LIN {X 0,Y 390.064,Z 239.895,A -85,B 0,C 180,E1 -11765.518,E2 -11765.518} C_VEL
LIN {X 0,Y 390.059,Z 239.898,A -85,B 0,C 180,E1 -11768.878,E2 -11768.878} C_VEL
LIN {X 0,Y 390.13,Z 239.89,A -85,B 0,C 180,E1 -11772.167,E2 -11772.167} C_VEL
LIN {X 0,Y 390.147,Z 239.885,A -85,B 0,C 180,E1 -11775.392,E2 -11775.392} C_VEL
LIN {X 0,Y 390.15,Z 239.886,A -85,B 0,C 180,E1 -11778.571,E2 -11778.571} C_VEL
LIN {X 0,Y 390.259,Z 239.876,A -85,B 0,C 180,E1 -11782.086,E2 -11782.086} C_VEL
LIN {X 0,Y 390.199,Z 239.878,A -85,B 0,C 180,E1 -11784.833,E2 -11784.833} C_VEL
LIN {X 0,Y 390.407,Z 239.856,A -85,B 0,C 180,E1 -11787.937,E2 -11787.937} C_VEL
LIN {X 0,Y 390.295,Z 239.866,A -85,B 0,C 180,E1 -11791.032,E2 -11791.032} C_VEL
LIN {X 0,Y 390.263,Z 239.871,A -85,B 0,C 180,E1 -11793.097,E2 -11793.097} C_VEL
LIN {X 0,Y 390.058,Z 240.018,A -85,B 0,C 180,E1 -11795.428,E2 -11795.428} C_VEL
LIN {X 0,Y 389.833,Z 246.867,A -85,B 0,C 180,E1 -11798.815,E2 -11798.815} C_VEL
LIN {X 0,Y 389.754,Z 254.263,A -85,B 0,C 180,E1 -11802.497,E2 -11802.497} C_VEL
LIN {X 0,Y 389.562,Z 261.72,A -85,B 0,C 180,E1 -11806.238,E2 -11806.238} C_VEL
LIN {X 0,Y 389.404,Z 267.139,A -85,B 0,C 180,E1 -11808.957,E2 -11808.957} C_VEL
LIN {X 0,Y 389.348,Z 274.683,A -85,B 0,C 180,E1 -11812.716,E2 -11812.716} C_VEL
LIN {X 0,Y 391.468,Z 286.466,A -85,B 0,C 180,E1 -11813.264,E2 -11813.264} C_VEL
LIN {X 0,Y 391.781,Z 288.367,A -85,B 0,C 180,E1 -11813.369,E2 -11813.369} C_VEL
LIN {X 0,Y 391.491,Z 292.048,A -85,B 0,C 180,E1 -11813.57,E2 -11813.57} C_VEL
LIN {X 0,Y 390.029,Z 295.619,A -85,B 0,C 180,E1 -11813.741,E2 -11813.741} C_VEL
LIN {X 0,Y 385.706,Z 303.652,A -85,B 0,C 180,E1 -11814.196,E2 -11814.196} C_VEL
LIN {X 0,Y 384.887,Z 307.067,A -85,B 0,C 180,E1 -11814.478,E2 -11814.478} C_VEL
LIN {X 0,Y 384.4,Z 315.281,A -85,B 0,C 180,E1 -11815.3,E2 -11815.3} C_VEL
LIN {X 0,Y 383.946,Z 322.929,A -85,B 0,C 180,E1 -11816.242,E2 -11816.242} C_VEL
LIN {X 0,Y 383.463,Z 329.813,A -85,B 0,C 180,E1 -11817.271,E2 -11817.271} C_VEL
LIN {X 0,Y 382.862,Z 337.958,A -85,B 0,C 180,E1 -11818.807,E2 -11818.807} C_VEL
LIN {X 0,Y 382.577,Z 341.952,A -85,B 0,C 180,E1 -11819.735,E2 -11819.735} C_VEL
LIN {X 0,Y 382.282,Z 346.3,A -85,B 0,C 180,E1 -11820.982,E2 -11820.982} C_VEL
LIN {X 0,Y 382.017,Z 349.759,A -85,B 0,C 180,E1 -11822.243,E2 -11822.243} C_VEL
LIN {X 0,Y 381.771,Z 353.226,A -85,B 0,C 180,E1 -11824.064,E2 -11824.064} C_VEL
LIN {X 0,Y 381.621,Z 355.211,A -85,B 0,C 180,E1 -11825.873,E2 -11825.873} C_VEL
LIN {X 0,Y 381.614,Z 355.585,A -85,B 0,C 180,E1 -11827.635,E2 -11827.635} C_VEL
LIN {X 0,Y 381.705,Z 354.659,A -85,B 0,C 180,E1 -11829.348,E2 -11829.348} C_VEL
LIN {X 0,Y 381.96,Z 352.506,A -85,B 0,C 180,E1 -11831.027,E2 -11831.027} C_VEL
LIN {X 0,Y 382.337,Z 348.46,A -85,B 0,C 180,E1 -11832.853,E2 -11832.853} C_VEL
LIN {X 0,Y 382.689,Z 344.128,A -85,B 0,C 180,E1 -11834.256,E2 -11834.256} C_VEL
LIN {X 0,Y 383.166,Z 338.499,A -85,B 0,C 180,E1 -11835.671,E2 -11835.671} C_VEL
LIN {X 0,Y 383.79,Z 331.204,A -85,B 0,C 180,E1 -11837.095,E2 -11837.095} C_VEL
LIN {X 0,Y 384.405,Z 323.923,A -85,B 0,C 180,E1 -11838.211,E2 -11838.211} C_VEL
LIN {X 0,Y 384.9,Z 317.284,A -85,B 0,C 180,E1 -11839.056,E2 -11839.056} C_VEL
LIN {X 0,Y 385.39,Z 310.045,A -85,B 0,C 180,E1 -11839.823,E2 -11839.823} C_VEL
LIN {X 0,Y 385.892,Z 301.292,A -85,B 0,C 180,E1 -11840.573,E2 -11840.573} C_VEL
LIN {X 0,Y 386.17,Z 294.889,A -85,B 0,C 180,E1 -11841.022,E2 -11841.022} C_VEL
LIN {X 0,Y 384.636,Z 285.462,A -85,B 0,C 180,E1 -11841.622,E2 -11841.622} C_VEL
LIN {X 0,Y 382.519,Z 275.828,A -85,B 0,C 180,E1 -11842.116,E2 -11842.116} C_VEL
LIN {X 0,Y 382.655,Z 268.589,A -85,B 0,C 180,E1 -11845.74,E2 -11845.74} C_VEL
LIN {X 0,Y 382.785,Z 261.93,A -85,B 0,C 180,E1 -11849.063,E2 -11849.063} C_VEL
LIN {X 0,Y 382.923,Z 256.534,A -85,B 0,C 180,E1 -11851.76,E2 -11851.76} C_VEL
LIN {X 0,Y 383.075,Z 248.588,A -85,B 0,C 180,E1 -11855.619,E2 -11855.619} C_VEL
LIN {X 0,Y 383.186,Z 242.55,A -85,B 0,C 180,E1 -11858.48,E2 -11858.48} C_VEL
LIN {X 0,Y 383.007,Z 240.78,A -85,B 0,C 180,E1 -11859.363,E2 -11859.363} C_VEL
LIN {X 0,Y 383.107,Z 240.766,A -85,B 0,C 180,E1 -11862.931,E2 -11862.931} C_VEL
LIN {X 0,Y 383.128,Z 240.763,A -85,B 0,C 180,E1 -11866.464,E2 -11866.464} C_VEL
LIN {X 0,Y 383.154,Z 240.762,A -85,B 0,C 180,E1 -11870.498,E2 -11870.498} C_VEL
LIN {X 0,Y 383.246,Z 240.748,A -85,B 0,C 180,E1 -11873.683,E2 -11873.683} C_VEL
LIN {X 0,Y 383.388,Z 240.73,A -85,B 0,C 180,E1 -11877.899,E2 -11877.899} C_VEL
LIN {X 0,Y 383.52,Z 240.713,A -85,B 0,C 180,E1 -11880,E2 -11880} C_VEL
LIN {X 0,Y 383.248,Z 240.747,A -85,B 0,C 180,E1 -11883.154,E2 -11883.154} C_VEL
LIN {X 0,Y 383.258,Z 240.745,A -85,B 0,C 180,E1 -11886.317,E2 -11886.317} C_VEL
LIN {X 0,Y 383.153,Z 240.76,A -85,B 0,C 180,E1 -11889.502,E2 -11889.502} C_VEL
LIN {X 0,Y 383.127,Z 240.76,A -85,B 0,C 180,E1 -11893.536,E2 -11893.536} C_VEL
LIN {X 0,Y 383.097,Z 240.766,A -85,B 0,C 180,E1 -11897.454,E2 -11897.454} C_VEL
LIN {X 0,Y 383.03,Z 240.773,A -85,B 0,C 180,E1 -11900.647,E2 -11900.647} C_VEL
LIN {X 0,Y 383.023,Z 240.774,A -85,B 0,C 180,E1 -11903.808,E2 -11903.808} C_VEL
LIN {X 0,Y 383.08,Z 240.768,A -85,B 0,C 180,E1 -11906.123,E2 -11906.123} C_VEL
LIN {X 0,Y 383.042,Z 240.774,A -85,B 0,C 180,E1 -11908.493,E2 -11908.493} C_VEL
LIN {X 0,Y 383.011,Z 240.774,A -85,B 0,C 180,E1 -11912.15,E2 -11912.15} C_VEL
LIN {X 0,Y 383.019,Z 240.773,A -85,B 0,C 180,E1 -11914.668,E2 -11914.668} C_VEL
LIN {X 0,Y 383.001,Z 240.777,A -85,B 0,C 180,E1 -11917.904,E2 -11917.904} C_VEL
LIN {X 0,Y 382.985,Z 240.78,A -85,B 0,C 180,E1 -11921.347,E2 -11921.347} C_VEL
LIN {X 0,Y 382.997,Z 240.779,A -85,B 0,C 180,E1 -11924.303,E2 -11924.303} C_VEL
LIN {X 0,Y 383.08,Z 240.924,A -85,B 0,C 180,E1 -11926.817,E2 -11926.817} C_VEL
LIN {X 0,Y 384.123,Z 247.016,A -85,B 0,C 180,E1 -11930.214,E2 -11930.214} C_VEL
LIN {X 0,Y 384.988,Z 252.135,A -85,B 0,C 180,E1 -11932.957,E2 -11932.957} C_VEL
LIN {X 0,Y 384.935,Z 256.673,A -85,B 0,C 180,E1 -11935.245,E2 -11935.245} C_VEL
LIN {X 0,Y 384.304,Z 262.28,A -85,B 0,C 180,E1 -11937.971,E2 -11937.971} C_VEL
LIN {X 0,Y 383.595,Z 269.862,A -85,B 0,C 180,E1 -11941.574,E2 -11941.574} C_VEL
LIN {X 0,Y 383.025,Z 277.322,A -85,B 0,C 180,E1 -11945.038,E2 -11945.038} C_VEL
LIN {X 0,Y 382.517,Z 284.78,A -85,B 0,C 180,E1 -11948.441,E2 -11948.441} C_VEL
LIN {X 0,Y 382.133,Z 292.511,A -85,B 0,C 180,E1 -11951.92,E2 -11951.92} C_VEL
LIN {X 0,Y 383.821,Z 306.099,A -85,B 0,C 180,E1 -11952.506,E2 -11952.506} C_VEL
LIN {X 0,Y 385.335,Z 319.619,A -85,B 0,C 180,E1 -11953.306,E2 -11953.306} C_VEL
LIN {X 0,Y 385.814,Z 325.668,A -85,B 0,C 180,E1 -11953.736,E2 -11953.736} C_VEL
LIN {X 0,Y 384.998,Z 337.028,A -85,B 0,C 180,E1 -11954.651,E2 -11954.651} C_VEL
LIN {X 0,Y 384.223,Z 347.555,A -85,B 0,C 180,E1 -11955.712,E2 -11955.712} C_VEL
LIN {X 0,Y 383.503,Z 358.111,A -85,B 0,C 180,E1 -11957.027,E2 -11957.027} C_VEL
LIN {X 0,Y 382.872,Z 366.826,A -85,B 0,C 180,E1 -11958.351,E2 -11958.351} C_VEL
LIN {X 0,Y 382.323,Z 375.346,A -85,B 0,C 180,E1 -11959.943,E2 -11959.943} C_VEL
LIN {X 0,Y 382.009,Z 382.192,A -85,B 0,C 180,E1 -11961.537,E2 -11961.537} C_VEL
LIN {X 0,Y 381.83,Z 387.648,A -85,B 0,C 180,E1 -11963.129,E2 -11963.129} C_VEL
LIN {X 0,Y 381.746,Z 391.876,A -85,B 0,C 180,E1 -11964.719,E2 -11964.719} C_VEL
LIN {X 0,Y 381.68,Z 394.089,A -85,B 0,C 180,E1 -11965.776,E2 -11965.776} C_VEL
LIN {X 0,Y 381.711,Z 395.798,A -85,B 0,C 180,E1 -11966.834,E2 -11966.834} C_VEL
LIN {X 0,Y 381.784,Z 397.076,A -85,B 0,C 180,E1 -11967.89,E2 -11967.89} C_VEL
LIN {X 0,Y 381.741,Z 397.928,A -85,B 0,C 180,E1 -11968.945,E2 -11968.945} C_VEL
LIN {X 0,Y 381.728,Z 398.341,A -85,B 0,C 180,E1 -11970,E2 -11970} C_VEL
LIN {X 0,Y 381.722,Z 398.306,A -85,B 0,C 180,E1 -11971.055,E2 -11971.055} C_VEL
LIN {X 0,Y 381.745,Z 397.863,A -85,B 0,C 180,E1 -11972.11,E2 -11972.11} C_VEL
LIN {X 0,Y 381.625,Z 397.006,A -85,B 0,C 180,E1 -11973.167,E2 -11973.167} C_VEL
LIN {X 0,Y 381.653,Z 395.705,A -85,B 0,C 180,E1 -11974.224,E2 -11974.224} C_VEL
LIN {X 0,Y 381.69,Z 392.269,A -85,B 0,C 180,E1 -11976.122,E2 -11976.122} C_VEL
LIN {X 0,Y 381.912,Z 387.634,A -85,B 0,C 180,E1 -11977.933,E2 -11977.933} C_VEL
LIN {X 0,Y 382.365,Z 381.352,A -85,B 0,C 180,E1 -11979.789,E2 -11979.789} C_VEL
LIN {X 0,Y 383.047,Z 373.281,A -85,B 0,C 180,E1 -11981.644,E2 -11981.644} C_VEL
LIN {X 0,Y 384.014,Z 364.697,A -85,B 0,C 180,E1 -11983.225,E2 -11983.225} C_VEL
LIN {X 0,Y 384.9,Z 355.689,A -85,B 0,C 180,E1 -11984.592,E2 -11984.592} C_VEL
LIN {X 0,Y 386.269,Z 344.532,A -85,B 0,C 180,E1 -11985.974,E2 -11985.974} C_VEL
LIN {X 0,Y 387.633,Z 332.921,A -85,B 0,C 180,E1 -11987.135,E2 -11987.135} C_VEL
LIN {X 0,Y 388.132,Z 325.333,A -85,B 0,C 180,E1 -11987.792,E2 -11987.792} C_VEL
LIN {X 0,Y 387.528,Z 312.932,A -85,B 0,C 180,E1 -11988.781,E2 -11988.781} C_VEL
LIN {X 0,Y 385.488,Z 300.133,A -85,B 0,C 180,E1 -11989.711,E2 -11989.711} C_VEL
LIN {X 0,Y 382.494,Z 287.785,A -85,B 0,C 180,E1 -11990.559,E2 -11990.559} C_VEL
LIN {X 0,Y 382.921,Z 280.937,A -85,B 0,C 180,E1 -11993.815,E2 -11993.815} C_VEL
LIN {X 0,Y 383.578,Z 274.157,A -85,B 0,C 180,E1 -11997.262,E2 -11997.262} C_VEL
LIN {X 0,Y 384.413,Z 267.801,A -85,B 0,C 180,E1 -12000.791,E2 -12000.791} C_VEL
LIN {X 0,Y 385.452,Z 262.026,A -85,B 0,C 180,E1 -12004.418,E2 -12004.418} C_VEL
LIN {X 0,Y 385.784,Z 258.61,A -85,B 0,C 180,E1 -12006.955,E2 -12006.955} C_VEL
LIN {X 0,Y 385.601,Z 255.652,A -85,B 0,C 180,E1 -12009.637,E2 -12009.637} C_VEL
LIN {X 0,Y 385.196,Z 253.221,A -85,B 0,C 180,E1 -12012.461,E2 -12012.461} C_VEL
LIN {X 0,Y 384.881,Z 251.375,A -85,B 0,C 180,E1 -12015.41,E2 -12015.41} C_VEL
LIN {X 0,Y 384.65,Z 250.149,A -85,B 0,C 180,E1 -12018.515,E2 -12018.515} C_VEL
LIN {X 0,Y 384.459,Z 249.598,A -85,B 0,C 180,E1 -12021.819,E2 -12021.819} C_VEL
LIN {X 0,Y 384.362,Z 249.644,A -85,B 0,C 180,E1 -12024.189,E2 -12024.189} C_VEL
LIN {X 0,Y 384.031,Z 250.218,A -85,B 0,C 180,E1 -12027.334,E2 -12027.334} C_VEL
LIN {X 0,Y 383.652,Z 251.212,A -85,B 0,C 180,E1 -12030.356,E2 -12030.356} C_VEL
LIN {X 0,Y 383.284,Z 252.849,A -85,B 0,C 180,E1 -12033.96,E2 -12033.96} C_VEL
LIN {X 0,Y 382.967,Z 254.746,A -85,B 0,C 180,E1 -12037.333,E2 -12037.333} C_VEL
LIN {X 0,Y 382.794,Z 256.871,A -85,B 0,C 180,E1 -12040.633,E2 -12040.633} C_VEL
LIN {X 0,Y 383.82,Z 259.798,A -85,B 0,C 180,E1 -12040.87,E2 -12040.87} C_VEL
LIN {X 0,Y 387.985,Z 270.603,A -85,B 0,C 180,E1 -12041.849,E2 -12041.849} C_VEL
LIN {X 0,Y 390.513,Z 280.022,A -85,B 0,C 180,E1 -12042.712,E2 -12042.712} C_VEL
LIN {X 0,Y 390.497,Z 283.446,A -85,B 0,C 180,E1 -12042.977,E2 -12042.977} C_VEL
LIN {X 0,Y 389.314,Z 295.932,A -85,B 0,C 180,E1 -12044.029,E2 -12044.029} C_VEL
LIN {X 0,Y 388.056,Z 306.9,A -85,B 0,C 180,E1 -12045.178,E2 -12045.178} C_VEL
LIN {X 0,Y 386.93,Z 315.954,A -85,B 0,C 180,E1 -12046.342,E2 -12046.342} C_VEL
LIN {X 0,Y 385.714,Z 325.894,A -85,B 0,C 180,E1 -12047.905,E2 -12047.905} C_VEL
LIN {X 0,Y 384.598,Z 333.903,A -85,B 0,C 180,E1 -12049.471,E2 -12049.471} C_VEL
LIN {X 0,Y 383.857,Z 340.374,A -85,B 0,C 180,E1 -12051.047,E2 -12051.047} C_VEL
LIN {X 0,Y 383.015,Z 345.589,A -85,B 0,C 180,E1 -12052.62,E2 -12052.62} C_VEL
LIN {X 0,Y 382.778,Z 349.616,A -85,B 0,C 180,E1 -12054.204,E2 -12054.204} C_VEL
LIN {X 0,Y 382.457,Z 352.63,A -85,B 0,C 180,E1 -12055.785,E2 -12055.785} C_VEL
LIN {X 0,Y 382.34,Z 354.101,A -85,B 0,C 180,E1 -12056.839,E2 -12056.839} C_VEL
LIN {X 0,Y 382.016,Z 355.174,A -85,B 0,C 180,E1 -12057.891,E2 -12057.891} C_VEL
LIN {X 0,Y 381.771,Z 356.022,A -85,B 0,C 180,E1 -12060,E2 -12060} C_VEL
LIN {X 0,Y 381.76,Z 355.851,A -85,B 0,C 180,E1 -12061.055,E2 -12061.055} C_VEL
LIN {X 0,Y 381.827,Z 355.248,A -85,B 0,C 180,E1 -12062.11,E2 -12062.11} C_VEL
LIN {X 0,Y 381.849,Z 354.219,A -85,B 0,C 180,E1 -12063.165,E2 -12063.165} C_VEL
LIN {X 0,Y 381.825,Z 352.79,A -85,B 0,C 180,E1 -12064.222,E2 -12064.222} C_VEL
LIN {X 0,Y 382.002,Z 349.805,A -85,B 0,C 180,E1 -12065.808,E2 -12065.808} C_VEL
LIN {X 0,Y 382.153,Z 345.762,A -85,B 0,C 180,E1 -12067.397,E2 -12067.397} C_VEL
LIN {X 0,Y 382.544,Z 339.557,A -85,B 0,C 180,E1 -12069.251,E2 -12069.251} C_VEL
LIN {X 0,Y 382.976,Z 332.754,A -85,B 0,C 180,E1 -12070.842,E2 -12070.842} C_VEL
LIN {X 0,Y 383.602,Z 324.348,A -85,B 0,C 180,E1 -12072.432,E2 -12072.432} C_VEL
LIN {X 0,Y 384.278,Z 314.547,A -85,B 0,C 180,E1 -12073.924,E2 -12073.924} C_VEL
LIN {X 0,Y 384.893,Z 304.111,A -85,B 0,C 180,E1 -12075.218,E2 -12075.218} C_VEL
LIN {X 0,Y 385.693,Z 293.658,A -85,B 0,C 180,E1 -12076.27,E2 -12076.27} C_VEL
LIN {X 0,Y 386.513,Z 280.873,A -85,B 0,C 180,E1 -12077.289,E2 -12077.289} C_VEL
LIN {X 0,Y 386.737,Z 275.385,A -85,B 0,C 180,E1 -12077.655,E2 -12077.655} C_VEL
LIN {X 0,Y 384.045,Z 262.022,A -85,B 0,C 180,E1 -12078.479,E2 -12078.479} C_VEL
LIN {X 0,Y 381.923,Z 251.524,A -85,B 0,C 180,E1 -12078.994,E2 -12078.994} C_VEL
LIN {X 0,Y 381.915,Z 247.631,A -85,B 0,C 180,E1 -12082.734,E2 -12082.734} C_VEL
LIN {X 0,Y 382.077,Z 244.102,A -85,B 0,C 180,E1 -12086.197,E2 -12086.197} C_VEL
LIN {X 0,Y 382.103,Z 241.747,A -85,B 0,C 180,E1 -12088.569,E2 -12088.569} C_VEL
LIN {X 0,Y 382.166,Z 240.883,A -85,B 0,C 180,E1 -12089.771,E2 -12089.771} C_VEL
LIN {X 0,Y 382.621,Z 240.827,A -85,B 0,C 180,E1 -12093.439,E2 -12093.439} C_VEL
LIN {X 0,Y 382.905,Z 240.787,A -85,B 0,C 180,E1 -12096.138,E2 -12096.138} C_VEL
LIN {X 0,Y 382.996,Z 240.777,A -85,B 0,C 180,E1 -12098.602,E2 -12098.602} C_VEL
LIN {X 0,Y 382.985,Z 240.781,A -85,B 0,C 180,E1 -12101.348,E2 -12101.348} C_VEL
LIN {X 0,Y 382.999,Z 240.775,A -85,B 0,C 180,E1 -12104.303,E2 -12104.303} C_VEL
LIN {X 0,Y 383.014,Z 240.776,A -85,B 0,C 180,E1 -12107.24,E2 -12107.24} C_VEL
LIN {X 0,Y 382.988,Z 240.778,A -85,B 0,C 180,E1 -12110.419,E2 -12110.419} C_VEL
LIN {X 0,Y 383.016,Z 240.772,A -85,B 0,C 180,E1 -12114.043,E2 -12114.043} C_VEL
LIN {X 0,Y 382.989,Z 240.776,A -85,B 0,C 180,E1 -12117.578,E2 -12117.578} C_VEL
LIN {X 0,Y 382.988,Z 240.779,A -85,B 0,C 180,E1 -12120.299,E2 -12120.299} C_VEL
LIN {X 0,Y 383.046,Z 240.771,A -85,B 0,C 180,E1 -12124.032,E2 -12124.032} C_VEL
LIN {X 0,Y 382.995,Z 240.776,A -85,B 0,C 180,E1 -12127.334,E2 -12127.334} C_VEL
LIN {X 0,Y 383.062,Z 240.77,A -85,B 0,C 180,E1 -12130.716,E2 -12130.716} C_VEL
LIN {X 0,Y 383.084,Z 240.768,A -85,B 0,C 180,E1 -12134.027,E2 -12134.027} C_VEL
LIN {X 0,Y 383.14,Z 240.758,A -85,B 0,C 180,E1 -12137.284,E2 -12137.284} C_VEL
LIN {X 0,Y 383.146,Z 240.758,A -85,B 0,C 180,E1 -12140.498,E2 -12140.498} C_VEL
LIN {X 0,Y 383.234,Z 240.748,A -85,B 0,C 180,E1 -12143.683,E2 -12143.683} C_VEL
LIN {X 0,Y 383.371,Z 240.733,A -85,B 0,C 180,E1 -12147.899,E2 -12147.899} C_VEL
LIN {X 0,Y 383.266,Z 240.741,A -85,B 0,C 180,E1 -12151.051,E2 -12151.051} C_VEL
LIN {X 0,Y 383.381,Z 240.729,A -85,B 0,C 180,E1 -12152.101,E2 -12152.101} C_VEL
LIN {X 0,Y 383.049,Z 240.859,A -85,B 0,C 180,E1 -12155.329,E2 -12155.329} C_VEL
LIN {X 0,Y 382.786,Z 248.186,A -85,B 0,C 180,E1 -12158.978,E2 -12158.978} C_VEL
LIN {X 0,Y 382.71,Z 255.662,A -85,B 0,C 180,E1 -12162.73,E2 -12162.73} C_VEL
LIN {X 0,Y 382.488,Z 263.248,A -85,B 0,C 180,E1 -12166.547,E2 -12166.547} C_VEL
LIN {X 0,Y 382.329,Z 269.769,A -85,B 0,C 180,E1 -12169.838,E2 -12169.838} C_VEL
LIN {X 0,Y 382.277,Z 274.974,A -85,B 0,C 180,E1 -12172.461,E2 -12172.461} C_VEL
LIN {X 0,Y 384.76,Z 288.83,A -85,B 0,C 180,E1 -12173.151,E2 -12173.151} C_VEL
LIN {X 0,Y 385.45,Z 294.606,A -85,B 0,C 180,E1 -12173.524,E2 -12173.524} C_VEL
LIN {X 0,Y 384.959,Z 305.487,A -85,B 0,C 180,E1 -12174.332,E2 -12174.332} C_VEL
LIN {X 0,Y 384.887,Z 307.067,A -85,B 0,C 180,E1 -12174.478,E2 -12174.478} C_VEL
LIN {X 0,Y 384.053,Z 312.121,A -85,B 0,C 180,E1 -12174.932,E2 -12174.932} C_VEL
LIN {X 0,Y 380.771,Z 319.846,A -85,B 0,C 180,E1 -12175.722,E2 -12175.722} C_VEL
LIN {X 0,Y 377.398,Z 327.02,A -85,B 0,C 180,E1 -12176.621,E2 -12176.621} C_VEL
LIN {X 0,Y 376.404,Z 331.043,A -85,B 0,C 180,E1 -12177.26,E2 -12177.26} C_VEL
LIN {X 0,Y 375.794,Z 338.668,A -85,B 0,C 180,E1 -12178.761,E2 -12178.761} C_VEL
LIN {X 0,Y 375.433,Z 343.811,A -85,B 0,C 180,E1 -12180.05,E2 -12180.05} C_VEL
LIN {X 0,Y 375.038,Z 348.777,A -85,B 0,C 180,E1 -12181.648,E2 -12181.648} C_VEL
LIN {X 0,Y 374.854,Z 351.743,A -85,B 0,C 180,E1 -12182.937,E2 -12182.937} C_VEL
LIN {X 0,Y 374.647,Z 354.113,A -85,B 0,C 180,E1 -12184.371,E2 -12184.371} C_VEL
LIN {X 0,Y 374.521,Z 355.737,A -85,B 0,C 180,E1 -12186.205,E2 -12186.205} C_VEL
LIN {X 0,Y 374.526,Z 355.893,A -85,B 0,C 180,E1 -12187.988,E2 -12187.988} C_VEL
LIN {X 0,Y 374.662,Z 354.788,A -85,B 0,C 180,E1 -12189.727,E2 -12189.727} C_VEL
LIN {X 0,Y 374.975,Z 352.348,A -85,B 0,C 180,E1 -12191.435,E2 -12191.435} C_VEL
LIN {X 0,Y 375.173,Z 350.351,A -85,B 0,C 180,E1 -12192.406,E2 -12192.406} C_VEL
LIN {X 0,Y 375.501,Z 346.538,A -85,B 0,C 180,E1 -12193.829,E2 -12193.829} C_VEL
LIN {X 0,Y 375.968,Z 341.421,A -85,B 0,C 180,E1 -12195.263,E2 -12195.263} C_VEL
LIN {X 0,Y 376.486,Z 336.09,A -85,B 0,C 180,E1 -12196.457,E2 -12196.457} C_VEL
LIN {X 0,Y 377.021,Z 329.555,A -85,B 0,C 180,E1 -12197.651,E2 -12197.651} C_VEL
LIN {X 0,Y 377.644,Z 322.437,A -85,B 0,C 180,E1 -12198.711,E2 -12198.711} C_VEL
LIN {X 0,Y 378.38,Z 313.351,A -85,B 0,C 180,E1 -12199.805,E2 -12199.805} C_VEL
LIN {X 0,Y 378.987,Z 303.249,A -85,B 0,C 180,E1 -12200.734,E2 -12200.734} C_VEL
LIN {X 0,Y 379.367,Z 296.06,A -85,B 0,C 180,E1 -12201.263,E2 -12201.263} C_VEL
LIN {X 0,Y 377.864,Z 286.83,A -85,B 0,C 180,E1 -12201.877,E2 -12201.877} C_VEL
LIN {X 0,Y 375.685,Z 277.189,A -85,B 0,C 180,E1 -12202.387,E2 -12202.387} C_VEL
LIN {X 0,Y 375.496,Z 276.171,A -85,B 0,C 180,E1 -12202.449,E2 -12202.449} C_VEL
LIN {X 0,Y 375.629,Z 269.437,A -85,B 0,C 180,E1 -12205.854,E2 -12205.854} C_VEL
LIN {X 0,Y 375.802,Z 262.494,A -85,B 0,C 180,E1 -12209.346,E2 -12209.346} C_VEL
LIN {X 0,Y 375.977,Z 255.707,A -85,B 0,C 180,E1 -12212.744,E2 -12212.744} C_VEL
LIN {X 0,Y 376.168,Z 248.436,A -85,B 0,C 180,E1 -12216.273,E2 -12216.273} C_VEL
LIN {X 0,Y 376.135,Z 242.637,A -85,B 0,C 180,E1 -12219.106,E2 -12219.106} C_VEL
LIN {X 0,Y 375.989,Z 241.654,A -85,B 0,C 180,E1 -12219.626,E2 -12219.626} C_VEL
LIN {X 0,Y 376.053,Z 241.645,A -85,B 0,C 180,E1 -12222.601,E2 -12222.601} C_VEL
LIN {X 0,Y 376.092,Z 241.639,A -85,B 0,C 180,E1 -12226.342,E2 -12226.342} C_VEL
LIN {X 0,Y 376.121,Z 241.637,A -85,B 0,C 180,E1 -12230.318,E2 -12230.318} C_VEL
LIN {X 0,Y 376.204,Z 241.625,A -85,B 0,C 180,E1 -12233.564,E2 -12233.564} C_VEL
LIN {X 0,Y 376.354,Z 241.606,A -85,B 0,C 180,E1 -12237.859,E2 -12237.859} C_VEL
LIN {X 0,Y 376.49,Z 241.589,A -85,B 0,C 180,E1 -12240,E2 -12240} C_VEL
LIN {X 0,Y 376.186,Z 241.627,A -85,B 0,C 180,E1 -12243.213,E2 -12243.213} C_VEL
LIN {X 0,Y 376.216,Z 241.623,A -85,B 0,C 180,E1 -12246.435,E2 -12246.435} C_VEL
LIN {X 0,Y 376.121,Z 241.637,A -85,B 0,C 180,E1 -12249.681,E2 -12249.681} C_VEL
LIN {X 0,Y 376.091,Z 241.636,A -85,B 0,C 180,E1 -12253.658,E2 -12253.658} C_VEL
LIN {X 0,Y 376.045,Z 241.645,A -85,B 0,C 180,E1 -12257.607,E2 -12257.607} C_VEL
LIN {X 0,Y 375.98,Z 241.651,A -85,B 0,C 180,E1 -12260.832,E2 -12260.832} C_VEL
LIN {X 0,Y 375.988,Z 241.649,A -85,B 0,C 180,E1 -12264.282,E2 -12264.282} C_VEL
LIN {X 0,Y 376.021,Z 241.644,A -85,B 0,C 180,E1 -12266.652,E2 -12266.652} C_VEL
LIN {X 0,Y 375.972,Z 241.651,A -85,B 0,C 180,E1 -12269.079,E2 -12269.079} C_VEL
LIN {X 0,Y 375.95,Z 241.655,A -85,B 0,C 180,E1 -12272.828,E2 -12272.828} C_VEL
LIN {X 0,Y 375.959,Z 241.653,A -85,B 0,C 180,E1 -12275.415,E2 -12275.415} C_VEL
LIN {X 0,Y 375.976,Z 241.654,A -85,B 0,C 180,E1 -12278.271,E2 -12278.271} C_VEL
LIN {X 0,Y 375.936,Z 241.657,A -85,B 0,C 180,E1 -12281.601,E2 -12281.601} C_VEL
LIN {X 0,Y 375.928,Z 241.661,A -85,B 0,C 180,E1 -12285.269,E2 -12285.269} C_VEL
LIN {X 0,Y 376.035,Z 241.86,A -85,B 0,C 180,E1 -12286.63,E2 -12286.63} C_VEL
LIN {X 0,Y 377.007,Z 247.483,A -85,B 0,C 180,E1 -12289.845,E2 -12289.845} C_VEL
LIN {X 0,Y 377.986,Z 253.43,A -85,B 0,C 180,E1 -12293.084,E2 -12293.084} C_VEL
LIN {X 0,Y 377.933,Z 256.968,A -85,B 0,C 180,E1 -12294.907,E2 -12294.907} C_VEL
LIN {X 0,Y 377.263,Z 263.047,A -85,B 0,C 180,E1 -12297.932,E2 -12297.932} C_VEL
LIN {X 0,Y 376.602,Z 269.964,A -85,B 0,C 180,E1 -12301.294,E2 -12301.294} C_VEL
LIN {X 0,Y 375.931,Z 278.047,A -85,B 0,C 180,E1 -12305.125,E2 -12305.125} C_VEL
LIN {X 0,Y 375.422,Z 285.482,A -85,B 0,C 180,E1 -12308.59,E2 -12308.59} C_VEL
LIN {X 0,Y 375.062,Z 292.213,A -85,B 0,C 180,E1 -12311.686,E2 -12311.686} C_VEL
LIN {X 0,Y 376.724,Z 305.829,A -85,B 0,C 180,E1 -12312.288,E2 -12312.288} C_VEL
LIN {X 0,Y 378.24,Z 319.594,A -85,B 0,C 180,E1 -12313.123,E2 -12313.123} C_VEL
LIN {X 0,Y 378.798,Z 325.628,A -85,B 0,C 180,E1 -12313.564,E2 -12313.564} C_VEL
LIN {X 0,Y 377.968,Z 336.889,A -85,B 0,C 180,E1 -12314.497,E2 -12314.497} C_VEL
LIN {X 0,Y 377.184,Z 347.419,A -85,B 0,C 180,E1 -12315.587,E2 -12315.587} C_VEL
LIN {X 0,Y 376.536,Z 356.896,A -85,B 0,C 180,E1 -12316.783,E2 -12316.783} C_VEL
LIN {X 0,Y 375.879,Z 365.733,A -85,B 0,C 180,E1 -12318.131,E2 -12318.131} C_VEL
LIN {X 0,Y 375.259,Z 374.406,A -85,B 0,C 180,E1 -12319.751,E2 -12319.751} C_VEL
LIN {X 0,Y 374.946,Z 381.347,A -85,B 0,C 180,E1 -12321.376,E2 -12321.376} C_VEL
LIN {X 0,Y 374.748,Z 386.89,A -85,B 0,C 180,E1 -12322.998,E2 -12322.998} C_VEL
LIN {X 0,Y 374.662,Z 391.201,A -85,B 0,C 180,E1 -12324.618,E2 -12324.618} C_VEL
LIN {X 0,Y 374.614,Z 393.459,A -85,B 0,C 180,E1 -12325.696,E2 -12325.696} C_VEL
LIN {X 0,Y 374.62,Z 395.231,A -85,B 0,C 180,E1 -12326.774,E2 -12326.774} C_VEL
LIN {X 0,Y 374.717,Z 396.542,A -85,B 0,C 180,E1 -12327.85,E2 -12327.85} C_VEL
LIN {X 0,Y 374.672,Z 397.424,A -85,B 0,C 180,E1 -12328.925,E2 -12328.925} C_VEL
LIN {X 0,Y 374.657,Z 397.892,A -85,B 0,C 180,E1 -12330,E2 -12330} C_VEL
LIN {X 0,Y 374.654,Z 397.897,A -85,B 0,C 180,E1 -12331.075,E2 -12331.075} C_VEL
LIN {X 0,Y 374.643,Z 397.482,A -85,B 0,C 180,E1 -12332.15,E2 -12332.15} C_VEL
LIN {X 0,Y 374.534,Z 396.654,A -85,B 0,C 180,E1 -12333.227,E2 -12333.227} C_VEL
LIN {X 0,Y 374.577,Z 395.417,A -85,B 0,C 180,E1 -12334.304,E2 -12334.304} C_VEL
LIN {X 0,Y 374.586,Z 392.413,A -85,B 0,C 180,E1 -12336.071,E2 -12336.071} C_VEL
LIN {X 0,Y 374.768,Z 388.991,A -85,B 0,C 180,E1 -12337.543,E2 -12337.543} C_VEL
LIN {X 0,Y 375.087,Z 384.184,A -85,B 0,C 180,E1 -12339.164,E2 -12339.164} C_VEL
LIN {X 0,Y 375.702,Z 377.011,A -85,B 0,C 180,E1 -12341.055,E2 -12341.055} C_VEL
LIN {X 0,Y 376.668,Z 369.381,A -85,B 0,C 180,E1 -12342.664,E2 -12342.664} C_VEL
LIN {X 0,Y 377.508,Z 360.595,A -85,B 0,C 180,E1 -12344.198,E2 -12344.198} C_VEL
LIN {X 0,Y 378.894,Z 349.619,A -85,B 0,C 180,E1 -12345.74,E2 -12345.74} C_VEL
LIN {X 0,Y 380.406,Z 338.026,A -85,B 0,C 180,E1 -12347.055,E2 -12347.055} C_VEL
LIN {X 0,Y 381.526,Z 326.689,A -85,B 0,C 180,E1 -12348.111,E2 -12348.111} C_VEL
LIN {X 0,Y 381.031,Z 314.451,A -85,B 0,C 180,E1 -12349.15,E2 -12349.15} C_VEL
LIN {X 0,Y 379.107,Z 301.802,A -85,B 0,C 180,E1 -12350.14,E2 -12350.14} C_VEL
LIN {X 0,Y 376.206,Z 290.22,A -85,B 0,C 180,E1 -12351.001,E2 -12351.001} C_VEL
LIN {X 0,Y 375.53,Z 287.172,A -85,B 0,C 180,E1 -12351.217,E2 -12351.217} C_VEL
LIN {X 0,Y 376.066,Z 279.805,A -85,B 0,C 180,E1 -12354.866,E2 -12354.866} C_VEL
LIN {X 0,Y 376.662,Z 274.263,A -85,B 0,C 180,E1 -12357.805,E2 -12357.805} C_VEL
LIN {X 0,Y 377.582,Z 268.038,A -85,B 0,C 180,E1 -12361.411,E2 -12361.411} C_VEL
LIN {X 0,Y 378.27,Z 264.222,A -85,B 0,C 180,E1 -12363.875,E2 -12363.875} C_VEL
LIN {X 0,Y 378.798,Z 260.73,A -85,B 0,C 180,E1 -12366.421,E2 -12366.421} C_VEL
LIN {X 0,Y 378.711,Z 257.685,A -85,B 0,C 180,E1 -12369.122,E2 -12369.122} C_VEL
LIN {X 0,Y 378.329,Z 255.129,A -85,B 0,C 180,E1 -12372.007,E2 -12372.007} C_VEL
LIN {X 0,Y 377.995,Z 253.131,A -85,B 0,C 180,E1 -12375.047,E2 -12375.047} C_VEL
LIN {X 0,Y 377.747,Z 251.827,A -85,B 0,C 180,E1 -12378.091,E2 -12378.091} C_VEL
LIN {X 0,Y 377.533,Z 251.15,A -85,B 0,C 180,E1 -12381.432,E2 -12381.432} C_VEL
LIN {X 0,Y 377.373,Z 251.16,A -85,B 0,C 180,E1 -12384.737,E2 -12384.737} C_VEL
LIN {X 0,Y 377.074,Z 251.603,A -85,B 0,C 180,E1 -12387.282,E2 -12387.282} C_VEL
LIN {X 0,Y 376.758,Z 252.336,A -85,B 0,C 180,E1 -12389.758,E2 -12389.758} C_VEL
LIN {X 0,Y 376.344,Z 253.823,A -85,B 0,C 180,E1 -12393.373,E2 -12393.373} C_VEL
LIN {X 0,Y 375.993,Z 255.674,A -85,B 0,C 180,E1 -12396.888,E2 -12396.888} C_VEL
LIN {X 0,Y 375.837,Z 257.545,A -85,B 0,C 180,E1 -12399.975,E2 -12399.975} C_VEL
LIN {X 0,Y 376.94,Z 260.579,A -85,B 0,C 180,E1 -12400.245,E2 -12400.245} C_VEL
LIN {X 0,Y 381.537,Z 272.393,A -85,B 0,C 180,E1 -12401.392,E2 -12401.392} C_VEL
LIN {X 0,Y 384.142,Z 281.948,A -85,B 0,C 180,E1 -12402.33,E2 -12402.33} C_VEL
LIN {X 0,Y 383.477,Z 291.138,A -85,B 0,C 180,E1 -12403.086,E2 -12403.086} C_VEL
LIN {X 0,Y 382.104,Z 303.135,A -85,B 0,C 180,E1 -12404.259,E2 -12404.259} C_VEL
LIN {X 0,Y 380.688,Z 313.843,A -85,B 0,C 180,E1 -12405.568,E2 -12405.568} C_VEL
LIN {X 0,Y 379.565,Z 322.67,A -85,B 0,C 180,E1 -12406.89,E2 -12406.89} C_VEL
LIN {X 0,Y 378.316,Z 331.347,A -85,B 0,C 180,E1 -12408.48,E2 -12408.48} C_VEL
LIN {X 0,Y 377.287,Z 338.4,A -85,B 0,C 180,E1 -12410.078,E2 -12410.078} C_VEL
LIN {X 0,Y 376.316,Z 344.872,A -85,B 0,C 180,E1 -12411.926,E2 -12411.926} C_VEL
LIN {X 0,Y 375.916,Z 349.222,A -85,B 0,C 180,E1 -12413.559,E2 -12413.559} C_VEL
LIN {X 0,Y 375.628,Z 351.479,A -85,B 0,C 180,E1 -12414.632,E2 -12414.632} C_VEL
LIN {X 0,Y 375.41,Z 353.312,A -85,B 0,C 180,E1 -12415.706,E2 -12415.706} C_VEL
LIN {X 0,Y 375.303,Z 354.73,A -85,B 0,C 180,E1 -12416.78,E2 -12416.78} C_VEL
LIN {X 0,Y 374.949,Z 355.721,A -85,B 0,C 180,E1 -12417.852,E2 -12417.852} C_VEL
LIN {X 0,Y 374.698,Z 356.472,A -85,B 0,C 180,E1 -12420,E2 -12420} C_VEL
LIN {X 0,Y 374.691,Z 356.242,A -85,B 0,C 180,E1 -12421.075,E2 -12421.075} C_VEL
LIN {X 0,Y 374.763,Z 355.563,A -85,B 0,C 180,E1 -12422.15,E2 -12422.15} C_VEL
LIN {X 0,Y 374.754,Z 354.487,A -85,B 0,C 180,E1 -12423.225,E2 -12423.225} C_VEL
LIN {X 0,Y 374.751,Z 353.008,A -85,B 0,C 180,E1 -12424.302,E2 -12424.302} C_VEL
LIN {X 0,Y 374.934,Z 349.927,A -85,B 0,C 180,E1 -12425.918,E2 -12425.918} C_VEL
LIN {X 0,Y 375.088,Z 345.783,A -85,B 0,C 180,E1 -12427.537,E2 -12427.537} C_VEL
LIN {X 0,Y 375.516,Z 339.421,A -85,B 0,C 180,E1 -12429.425,E2 -12429.425} C_VEL
LIN {X 0,Y 375.954,Z 332.499,A -85,B 0,C 180,E1 -12431.047,E2 -12431.047} C_VEL
LIN {X 0,Y 376.632,Z 323.946,A -85,B 0,C 180,E1 -12432.666,E2 -12432.666} C_VEL
LIN {X 0,Y 377.325,Z 313.609,A -85,B 0,C 180,E1 -12434.232,E2 -12434.232} C_VEL
LIN {X 0,Y 378.007,Z 303.309,A -85,B 0,C 180,E1 -12435.502,E2 -12435.502} C_VEL
LIN {X 0,Y 378.926,Z 291,A -85,B 0,C 180,E1 -12436.707,E2 -12436.707} C_VEL
LIN {X 0,Y 379.684,Z 278.602,A -85,B 0,C 180,E1 -12437.667,E2 -12437.667} C_VEL
LIN {X 0,Y 379.312,Z 274.155,A -85,B 0,C 180,E1 -12437.974,E2 -12437.974} C_VEL
LIN {X 0,Y 376.628,Z 260.635,A -85,B 0,C 180,E1 -12438.793,E2 -12438.793} C_VEL
LIN {X 0,Y 374.823,Z 251.878,A -85,B 0,C 180,E1 -12439.226,E2 -12439.226} C_VEL
LIN {X 0,Y 374.821,Z 248.978,A -85,B 0,C 180,E1 -12442.025,E2 -12442.025} C_VEL
LIN {X 0,Y 375.025,Z 245.044,A -85,B 0,C 180,E1 -12445.903,E2 -12445.903} C_VEL
LIN {X 0,Y 375.05,Z 241.847,A -85,B 0,C 180,E1 -12449.158,E2 -12449.158} C_VEL
LIN {X 0,Y 375.495,Z 241.712,A -85,B 0,C 180,E1 -12452.874,E2 -12452.874} C_VEL
LIN {X 0,Y 375.805,Z 241.676,A -85,B 0,C 180,E1 -12455.432,E2 -12455.432} C_VEL
LIN {X 0,Y 375.967,Z 241.651,A -85,B 0,C 180,E1 -12458.268,E2 -12458.268} C_VEL
LIN {X 0,Y 375.936,Z 241.657,A -85,B 0,C 180,E1 -12461.6,E2 -12461.6} C_VEL
LIN {X 0,Y 375.929,Z 241.659,A -85,B 0,C 180,E1 -12465.269,E2 -12465.269} C_VEL
LIN {X 0,Y 375.921,Z 241.658,A -85,B 0,C 180,E1 -12468.402,E2 -12468.402} C_VEL
LIN {X 0,Y 375.955,Z 241.651,A -85,B 0,C 180,E1 -12471.91,E2 -12471.91} C_VEL
LIN {X 0,Y 375.977,Z 241.65,A -85,B 0,C 180,E1 -12475.334,E2 -12475.334} C_VEL
LIN {X 0,Y 375.96,Z 241.655,A -85,B 0,C 180,E1 -12478.438,E2 -12478.438} C_VEL
LIN {X 0,Y 375.961,Z 241.654,A -85,B 0,C 180,E1 -12482.138,E2 -12482.138} C_VEL
LIN {X 0,Y 375.98,Z 241.653,A -85,B 0,C 180,E1 -12484.537,E2 -12484.537} C_VEL
LIN {X 0,Y 375.96,Z 241.655,A -85,B 0,C 180,E1 -12488.045,E2 -12488.045} C_VEL
LIN {X 0,Y 376.011,Z 241.646,A -85,B 0,C 180,E1 -12491.473,E2 -12491.473} C_VEL
LIN {X 0,Y 376.062,Z 241.64,A -85,B 0,C 180,E1 -12494.832,E2 -12494.832} C_VEL
LIN {X 0,Y 376.053,Z 241.644,A -85,B 0,C 180,E1 -12498.136,E2 -12498.136} C_VEL
LIN {X 0,Y 376.189,Z 241.627,A -85,B 0,C 180,E1 -12501.955,E2 -12501.955} C_VEL
LIN {X 0,Y 376.143,Z 241.629,A -85,B 0,C 180,E1 -12504.639,E2 -12504.639} C_VEL
LIN {X 0,Y 376.335,Z 241.61,A -85,B 0,C 180,E1 -12507.859,E2 -12507.859} C_VEL
LIN {X 0,Y 376.237,Z 241.617,A -85,B 0,C 180,E1 -12511.07,E2 -12511.07} C_VEL
LIN {X 0,Y 376.345,Z 241.605,A -85,B 0,C 180,E1 -12512.14,E2 -12512.14} C_VEL
LIN {X 0,Y 376.021,Z 241.713,A -85,B 0,C 180,E1 -12515.228,E2 -12515.228} C_VEL
LIN {X 0,Y 375.766,Z 249.518,A -85,B 0,C 180,E1 -12519.147,E2 -12519.147} C_VEL
LIN {X 0,Y 375.648,Z 257.071,A -85,B 0,C 180,E1 -12522.974,E2 -12522.974} C_VEL
LIN {X 0,Y 375.46,Z 263.683,A -85,B 0,C 180,E1 -12526.306,E2 -12526.306} C_VEL
LIN {X 0,Y 375.324,Z 269.221,A -85,B 0,C 180,E1 -12529.129,E2 -12529.129} C_VEL
LIN {X 0,Y 375.213,Z 275.304,A -85,B 0,C 180,E1 -12532.218,E2 -12532.218} C_VEL
LIN {X 0,Y 377.575,Z 288.303,A -85,B 0,C 180,E1 -12532.865,E2 -12532.865} C_VEL
LIN {X 0,Y 378.5,Z 295.099,A -85,B 0,C 180,E1 -12533.312,E2 -12533.312} C_VEL
LIN {X 0,Y 378.016,Z 306.027,A -85,B 0,C 180,E1 -12534.143,E2 -12534.143} C_VEL
LIN {X 0,Y 377.456,Z 315.348,A -85,B 0,C 180,E1 -12535.079,E2 -12535.079} C_VEL
LIN {X 0,Y 376.992,Z 322.647,A -85,B 0,C 180,E1 -12535.982,E2 -12535.982} C_VEL
LIN {X 0,Y 376.529,Z 328.914,A -85,B 0,C 180,E1 -12536.913,E2 -12536.913} C_VEL
LIN {X 0,Y 376.404,Z 331.043,A -85,B 0,C 180,E1 -12537.26,E2 -12537.26} C_VEL
LIN {X 0,Y 375.445,Z 334.831,A -85,B 0,C 180,E1 -12537.938,E2 -12537.938} C_VEL
LIN {X 0,Y 372.181,Z 340.524,A -85,B 0,C 180,E1 -12539.08,E2 -12539.08} C_VEL
LIN {X 0,Y 368.962,Z 345.441,A -85,B 0,C 180,E1 -12540.318,E2 -12540.318} C_VEL
LIN {X 0,Y 368.088,Z 347.947,A -85,B 0,C 180,E1 -12541.139,E2 -12541.139} C_VEL
LIN {X 0,Y 367.787,Z 351.881,A -85,B 0,C 180,E1 -12542.776,E2 -12542.776} C_VEL
LIN {X 0,Y 367.53,Z 354.918,A -85,B 0,C 180,E1 -12544.688,E2 -12544.688} C_VEL
LIN {X 0,Y 367.435,Z 356.227,A -85,B 0,C 180,E1 -12546.549,E2 -12546.549} C_VEL
LIN {X 0,Y 367.474,Z 356.2,A -85,B 0,C 180,E1 -12548.359,E2 -12548.359} C_VEL
LIN {X 0,Y 367.629,Z 354.871,A -85,B 0,C 180,E1 -12550.121,E2 -12550.121} C_VEL
LIN {X 0,Y 367.979,Z 352.14,A -85,B 0,C 180,E1 -12551.853,E2 -12551.853} C_VEL
LIN {X 0,Y 368.148,Z 350.484,A -85,B 0,C 180,E1 -12552.664,E2 -12552.664} C_VEL
LIN {X 0,Y 368.64,Z 345.271,A -85,B 0,C 180,E1 -12554.492,E2 -12554.492} C_VEL
LIN {X 0,Y 369.056,Z 340.79,A -85,B 0,C 180,E1 -12555.704,E2 -12555.704} C_VEL
LIN {X 0,Y 369.661,Z 334.97,A -85,B 0,C 180,E1 -12556.975,E2 -12556.975} C_VEL
LIN {X 0,Y 370.214,Z 328.711,A -85,B 0,C 180,E1 -12558.094,E2 -12558.094} C_VEL
LIN {X 0,Y 370.982,Z 320.635,A -85,B 0,C 180,E1 -12559.268,E2 -12559.268} C_VEL
LIN {X 0,Y 371.642,Z 311.867,A -85,B 0,C 180,E1 -12560.271,E2 -12560.271} C_VEL
LIN {X 0,Y 372.204,Z 302.966,A -85,B 0,C 180,E1 -12561.078,E2 -12561.078} C_VEL
LIN {X 0,Y 372.554,Z 297.446,A -85,B 0,C 180,E1 -12561.499,E2 -12561.499} C_VEL
LIN {X 0,Y 370.878,Z 287.217,A -85,B 0,C 180,E1 -12562.2,E2 -12562.2} C_VEL
LIN {X 0,Y 368.762,Z 277.982,A -85,B 0,C 180,E1 -12562.71,E2 -12562.71} C_VEL
LIN {X 0,Y 368.482,Z 276.506,A -85,B 0,C 180,E1 -12562.805,E2 -12562.805} C_VEL
LIN {X 0,Y 368.633,Z 269.399,A -85,B 0,C 180,E1 -12566.434,E2 -12566.434} C_VEL
LIN {X 0,Y 368.811,Z 262.967,A -85,B 0,C 180,E1 -12569.678,E2 -12569.678} C_VEL
LIN {X 0,Y 368.994,Z 256.903,A -85,B 0,C 180,E1 -12572.799,E2 -12572.799} C_VEL
LIN {X 0,Y 369.195,Z 249.523,A -85,B 0,C 180,E1 -12576.437,E2 -12576.437} C_VEL
LIN {X 0,Y 369.208,Z 244.507,A -85,B 0,C 180,E1 -12578.865,E2 -12578.865} C_VEL
LIN {X 0,Y 368.949,Z 242.53,A -85,B 0,C 180,E1 -12579.948,E2 -12579.948} C_VEL
LIN {X 0,Y 368.978,Z 242.525,A -85,B 0,C 180,E1 -12583.399,E2 -12583.399} C_VEL
LIN {X 0,Y 369.06,Z 242.514,A -85,B 0,C 180,E1 -12586.79,E2 -12586.79} C_VEL
LIN {X 0,Y 369.07,Z 242.515,A -85,B 0,C 180,E1 -12590.132,E2 -12590.132} C_VEL
LIN {X 0,Y 369.165,Z 242.502,A -85,B 0,C 180,E1 -12593.441,E2 -12593.441} C_VEL
LIN {X 0,Y 369.319,Z 242.482,A -85,B 0,C 180,E1 -12597.819,E2 -12597.819} C_VEL
LIN {X 0,Y 369.459,Z 242.465,A -85,B 0,C 180,E1 -12600,E2 -12600} C_VEL
LIN {X 0,Y 369.319,Z 242.482,A -85,B 0,C 180,E1 -12602.181,E2 -12602.181} C_VEL
LIN {X 0,Y 369.176,Z 242.5,A -85,B 0,C 180,E1 -12606.559,E2 -12606.559} C_VEL
LIN {X 0,Y 369.069,Z 242.514,A -85,B 0,C 180,E1 -12609.868,E2 -12609.868} C_VEL
LIN {X 0,Y 369.039,Z 242.515,A -85,B 0,C 180,E1 -12613.772,E2 -12613.772} C_VEL
LIN {X 0,Y 369.003,Z 242.522,A -85,B 0,C 180,E1 -12617.768,E2 -12617.768} C_VEL
LIN {X 0,Y 368.911,Z 242.531,A -85,B 0,C 180,E1 -12621.221,E2 -12621.221} C_VEL
LIN {X 0,Y 368.955,Z 242.526,A -85,B 0,C 180,E1 -12624.776,E2 -12624.776} C_VEL
LIN {X 0,Y 368.97,Z 242.523,A -85,B 0,C 180,E1 -12627.203,E2 -12627.203} C_VEL
LIN {X 0,Y 368.92,Z 242.529,A -85,B 0,C 180,E1 -12629.69,E2 -12629.69} C_VEL
LIN {X 0,Y 368.898,Z 242.533,A -85,B 0,C 180,E1 -12633.043,E2 -12633.043} C_VEL
LIN {X 0,Y 368.918,Z 242.531,A -85,B 0,C 180,E1 -12636.197,E2 -12636.197} C_VEL
LIN {X 0,Y 368.905,Z 242.533,A -85,B 0,C 180,E1 -12638.953,E2 -12638.953} C_VEL
LIN {X 0,Y 368.882,Z 242.535,A -85,B 0,C 180,E1 -12642.009,E2 -12642.009} C_VEL
LIN {X 0,Y 368.898,Z 242.536,A -85,B 0,C 180,E1 -12645.821,E2 -12645.821} C_VEL
LIN {X 0,Y 368.963,Z 242.662,A -85,B 0,C 180,E1 -12646.371,E2 -12646.371} C_VEL
LIN {X 0,Y 369.983,Z 248.495,A -85,B 0,C 180,E1 -12649.771,E2 -12649.771} C_VEL
LIN {X 0,Y 370.858,Z 253.819,A -85,B 0,C 180,E1 -12652.743,E2 -12652.743} C_VEL
LIN {X 0,Y 370.951,Z 257.247,A -85,B 0,C 180,E1 -12654.555,E2 -12654.555} C_VEL
LIN {X 0,Y 370.388,Z 262.555,A -85,B 0,C 180,E1 -12657.263,E2 -12657.263} C_VEL
LIN {X 0,Y 369.576,Z 270.095,A -85,B 0,C 180,E1 -12661.016,E2 -12661.016} C_VEL
LIN {X 0,Y 368.938,Z 277.517,A -85,B 0,C 180,E1 -12664.621,E2 -12664.621} C_VEL
LIN {X 0,Y 368.373,Z 284.914,A -85,B 0,C 180,E1 -12668.159,E2 -12668.159} C_VEL
LIN {X 0,Y 367.997,Z 291.889,A -85,B 0,C 180,E1 -12671.452,E2 -12671.452} C_VEL
LIN {X 0,Y 369.64,Z 305.606,A -85,B 0,C 180,E1 -12672.069,E2 -12672.069} C_VEL
LIN {X 0,Y 371.168,Z 319.481,A -85,B 0,C 180,E1 -12672.933,E2 -12672.933} C_VEL
LIN {X 0,Y 371.725,Z 327.298,A -85,B 0,C 180,E1 -12673.525,E2 -12673.525} C_VEL
LIN {X 0,Y 370.873,Z 338.073,A -85,B 0,C 180,E1 -12674.475,E2 -12674.475} C_VEL
LIN {X 0,Y 369.976,Z 349.297,A -85,B 0,C 180,E1 -12675.703,E2 -12675.703} C_VEL
LIN {X 0,Y 369.224,Z 359.441,A -85,B 0,C 180,E1 -12677.076,E2 -12677.076} C_VEL
LIN {X 0,Y 368.641,Z 367.754,A -85,B 0,C 180,E1 -12678.453,E2 -12678.453} C_VEL
LIN {X 0,Y 368.107,Z 375.922,A -85,B 0,C 180,E1 -12680.106,E2 -12680.106} C_VEL
LIN {X 0,Y 367.82,Z 382.513,A -85,B 0,C 180,E1 -12681.761,E2 -12681.761} C_VEL
LIN {X 0,Y 367.636,Z 387.727,A -85,B 0,C 180,E1 -12683.414,E2 -12683.414} C_VEL
LIN {X 0,Y 367.612,Z 391.736,A -85,B 0,C 180,E1 -12685.065,E2 -12685.065} C_VEL
LIN {X 0,Y 367.531,Z 394.639,A -85,B 0,C 180,E1 -12686.711,E2 -12686.711} C_VEL
LIN {X 0,Y 367.651,Z 395.994,A -85,B 0,C 180,E1 -12687.809,E2 -12687.809} C_VEL
LIN {X 0,Y 367.606,Z 396.912,A -85,B 0,C 180,E1 -12688.905,E2 -12688.905} C_VEL
LIN {X 0,Y 367.588,Z 397.417,A -85,B 0,C 180,E1 -12690,E2 -12690} C_VEL
LIN {X 0,Y 367.587,Z 397.487,A -85,B 0,C 180,E1 -12691.096,E2 -12691.096} C_VEL
LIN {X 0,Y 367.543,Z 397.104,A -85,B 0,C 180,E1 -12692.192,E2 -12692.192} C_VEL
LIN {X 0,Y 367.48,Z 395.116,A -85,B 0,C 180,E1 -12694.388,E2 -12694.388} C_VEL
LIN {X 0,Y 367.486,Z 392.505,A -85,B 0,C 180,E1 -12696.024,E2 -12696.024} C_VEL
LIN {X 0,Y 367.695,Z 388.835,A -85,B 0,C 180,E1 -12697.689,E2 -12697.689} C_VEL
LIN {X 0,Y 368.035,Z 384.119,A -85,B 0,C 180,E1 -12699.342,E2 -12699.342} C_VEL
LIN {X 0,Y 368.7,Z 377.112,A -85,B 0,C 180,E1 -12701.267,E2 -12701.267} C_VEL
LIN {X 0,Y 369.903,Z 368.229,A -85,B 0,C 180,E1 -12703.179,E2 -12703.179} C_VEL
LIN {X 0,Y 370.72,Z 360.188,A -85,B 0,C 180,E1 -12704.602,E2 -12704.602} C_VEL
LIN {X 0,Y 372.259,Z 349.273,A -85,B 0,C 180,E1 -12706.169,E2 -12706.169} C_VEL
LIN {X 0,Y 373.879,Z 337.797,A -85,B 0,C 180,E1 -12707.504,E2 -12707.504} C_VEL
LIN {X 0,Y 374.933,Z 328.178,A -85,B 0,C 180,E1 -12708.441,E2 -12708.441} C_VEL
LIN {X 0,Y 374.718,Z 317.421,A -85,B 0,C 180,E1 -12709.41,E2 -12709.41} C_VEL
LIN {X 0,Y 372.967,Z 304.388,A -85,B 0,C 180,E1 -12710.506,E2 -12710.506} C_VEL
LIN {X 0,Y 370.259,Z 292.965,A -85,B 0,C 180,E1 -12711.43,E2 -12711.43} C_VEL
LIN {X 0,Y 368.576,Z 286.505,A -85,B 0,C 180,E1 -12711.946,E2 -12711.946} C_VEL
LIN {X 0,Y 369.256,Z 278.747,A -85,B 0,C 180,E1 -12715.961,E2 -12715.961} C_VEL
LIN {X 0,Y 370.064,Z 272.319,A -85,B 0,C 180,E1 -12719.589,E2 -12719.589} C_VEL
LIN {X 0,Y 370.762,Z 268.313,A -85,B 0,C 180,E1 -12722.057,E2 -12722.057} C_VEL
LIN {X 0,Y 371.464,Z 264.593,A -85,B 0,C 180,E1 -12724.583,E2 -12724.583} C_VEL
LIN {X 0,Y 371.878,Z 261.235,A -85,B 0,C 180,E1 -12727.212,E2 -12727.212} C_VEL
LIN {X 0,Y 371.653,Z 258.348,A -85,B 0,C 180,E1 -12730.012,E2 -12730.012} C_VEL
LIN {X 0,Y 371.281,Z 255.99,A -85,B 0,C 180,E1 -12732.957,E2 -12732.957} C_VEL
LIN {X 0,Y 370.984,Z 254.202,A -85,B 0,C 180,E1 -12736.045,E2 -12736.045} C_VEL
LIN {X 0,Y 370.722,Z 253.047,A -85,B 0,C 180,E1 -12739.316,E2 -12739.316} C_VEL
LIN {X 0,Y 370.527,Z 252.57,A -85,B 0,C 180,E1 -12742.811,E2 -12742.811} C_VEL
LIN {X 0,Y 370.374,Z 252.685,A -85,B 0,C 180,E1 -12745.301,E2 -12745.301} C_VEL
LIN {X 0,Y 369.867,Z 253.503,A -85,B 0,C 180,E1 -12749.134,E2 -12749.134} C_VEL
LIN {X 0,Y 369.566,Z 254.362,A -85,B 0,C 180,E1 -12751.613,E2 -12751.613} C_VEL
LIN {X 0,Y 369.28,Z 255.422,A -85,B 0,C 180,E1 -12754.041,E2 -12754.041} C_VEL
LIN {X 0,Y 368.921,Z 257.287,A -85,B 0,C 180,E1 -12757.604,E2 -12757.604} C_VEL
LIN {X 0,Y 368.875,Z 258.336,A -85,B 0,C 180,E1 -12759.27,E2 -12759.27} C_VEL
LIN {X 0,Y 369.944,Z 261.232,A -85,B 0,C 180,E1 -12759.546,E2 -12759.546} C_VEL
LIN {X 0,Y 374.306,Z 271.722,A -85,B 0,C 180,E1 -12760.653,E2 -12760.653} C_VEL
LIN {X 0,Y 377.434,Z 282.088,A -85,B 0,C 180,E1 -12761.742,E2 -12761.742} C_VEL
LIN {X 0,Y 377.91,Z 284.31,A -85,B 0,C 180,E1 -12761.97,E2 -12761.97} C_VEL
LIN {X 0,Y 376.444,Z 297.899,A -85,B 0,C 180,E1 -12763.179,E2 -12763.179} C_VEL
LIN {X 0,Y 375.015,Z 308.597,A -85,B 0,C 180,E1 -12764.372,E2 -12764.372} C_VEL
LIN {X 0,Y 373.752,Z 317.456,A -85,B 0,C 180,E1 -12765.573,E2 -12765.573} C_VEL
LIN {X 0,Y 372.336,Z 327.225,A -85,B 0,C 180,E1 -12767.186,E2 -12767.186} C_VEL
LIN {X 0,Y 371.095,Z 335.103,A -85,B 0,C 180,E1 -12768.807,E2 -12768.807} C_VEL
LIN {X 0,Y 370.244,Z 340.549,A -85,B 0,C 180,E1 -12770.163,E2 -12770.163} C_VEL
LIN {X 0,Y 369.343,Z 345.862,A -85,B 0,C 180,E1 -12771.79,E2 -12771.79} C_VEL
LIN {X 0,Y 368.912,Z 350.04,A -85,B 0,C 180,E1 -12773.437,E2 -12773.437} C_VEL
LIN {X 0,Y 368.613,Z 352.235,A -85,B 0,C 180,E1 -12774.53,E2 -12774.53} C_VEL
LIN {X 0,Y 368.367,Z 354.013,A -85,B 0,C 180,E1 -12775.623,E2 -12775.623} C_VEL
LIN {X 0,Y 368.266,Z 355.346,A -85,B 0,C 180,E1 -12776.718,E2 -12776.718} C_VEL
LIN {X 0,Y 367.884,Z 356.274,A -85,B 0,C 180,E1 -12777.81,E2 -12777.81} C_VEL
LIN {X 0,Y 367.627,Z 356.922,A -85,B 0,C 180,E1 -12780,E2 -12780} C_VEL
LIN {X 0,Y 367.625,Z 356.603,A -85,B 0,C 180,E1 -12781.096,E2 -12781.096} C_VEL
LIN {X 0,Y 367.681,Z 355.871,A -85,B 0,C 180,E1 -12782.191,E2 -12782.191} C_VEL
LIN {X 0,Y 367.659,Z 354.745,A -85,B 0,C 180,E1 -12783.288,E2 -12783.288} C_VEL
LIN {X 0,Y 367.745,Z 352.236,A -85,B 0,C 180,E1 -12784.934,E2 -12784.934} C_VEL
LIN {X 0,Y 367.947,Z 347.697,A -85,B 0,C 180,E1 -12786.973,E2 -12786.973} C_VEL
LIN {X 0,Y 368.253,Z 342.25,A -85,B 0,C 180,E1 -12788.782,E2 -12788.782} C_VEL
LIN {X 0,Y 368.669,Z 335.915,A -85,B 0,C 180,E1 -12790.434,E2 -12790.434} C_VEL
LIN {X 0,Y 369.269,Z 328.068,A -85,B 0,C 180,E1 -12792.085,E2 -12792.085} C_VEL
LIN {X 0,Y 370.005,Z 318.268,A -85,B 0,C 180,E1 -12793.735,E2 -12793.735} C_VEL
LIN {X 0,Y 370.713,Z 308.08,A -85,B 0,C 180,E1 -12795.131,E2 -12795.131} C_VEL
LIN {X 0,Y 371.544,Z 297.097,A -85,B 0,C 180,E1 -12796.342,E2 -12796.342} C_VEL
LIN {X 0,Y 372.4,Z 284.784,A -85,B 0,C 180,E1 -12797.434,E2 -12797.434} C_VEL
LIN {X 0,Y 372.624,Z 276.549,A -85,B 0,C 180,E1 -12798.028,E2 -12798.028} C_VEL
LIN {X 0,Y 370.002,Z 263.278,A -85,B 0,C 180,E1 -12798.892,E2 -12798.892} C_VEL
LIN {X 0,Y 367.77,Z 252.223,A -85,B 0,C 180,E1 -12799.465,E2 -12799.465} C_VEL
LIN {X 0,Y 367.799,Z 247.943,A -85,B 0,C 180,E1 -12803.658,E2 -12803.658} C_VEL
LIN {X 0,Y 367.941,Z 245.464,A -85,B 0,C 180,E1 -12806.136,E2 -12806.136} C_VEL
LIN {X 0,Y 367.989,Z 243.119,A -85,B 0,C 180,E1 -12808.534,E2 -12808.534} C_VEL
LIN {X 0,Y 368.061,Z 242.64,A -85,B 0,C 180,E1 -12809.766,E2 -12809.766} C_VEL
LIN {X 0,Y 368.537,Z 242.581,A -85,B 0,C 180,E1 -12813.575,E2 -12813.575} C_VEL
LIN {X 0,Y 368.856,Z 242.539,A -85,B 0,C 180,E1 -12816.846,E2 -12816.846} C_VEL
LIN {X 0,Y 368.912,Z 242.53,A -85,B 0,C 180,E1 -12820.37,E2 -12820.37} C_VEL
LIN {X 0,Y 368.886,Z 242.534,A -85,B 0,C 180,E1 -12823.616,E2 -12823.616} C_VEL
LIN {X 0,Y 368.888,Z 242.535,A -85,B 0,C 180,E1 -12826.696,E2 -12826.696} C_VEL
LIN {X 0,Y 368.887,Z 242.532,A -85,B 0,C 180,E1 -12829.648,E2 -12829.648} C_VEL
LIN {X 0,Y 368.898,Z 242.533,A -85,B 0,C 180,E1 -12833.146,E2 -12833.146} C_VEL
LIN {X 0,Y 368.898,Z 242.534,A -85,B 0,C 180,E1 -12836.462,E2 -12836.462} C_VEL
LIN {X 0,Y 368.933,Z 242.529,A -85,B 0,C 180,E1 -12839.046,E2 -12839.046} C_VEL
LIN {X 0,Y 368.902,Z 242.534,A -85,B 0,C 180,E1 -12842.791,E2 -12842.791} C_VEL
LIN {X 0,Y 368.932,Z 242.53,A -85,B 0,C 180,E1 -12846.119,E2 -12846.119} C_VEL
LIN {X 0,Y 368.94,Z 242.529,A -85,B 0,C 180,E1 -12849.947,E2 -12849.947} C_VEL
LIN {X 0,Y 368.979,Z 242.521,A -85,B 0,C 180,E1 -12853.399,E2 -12853.399} C_VEL
LIN {X 0,Y 369.061,Z 242.512,A -85,B 0,C 180,E1 -12856.79,E2 -12856.79} C_VEL
LIN {X 0,Y 369.066,Z 242.515,A -85,B 0,C 180,E1 -12860.131,E2 -12860.131} C_VEL
LIN {X 0,Y 369.156,Z 242.501,A -85,B 0,C 180,E1 -12863.441,E2 -12863.441} C_VEL
LIN {X 0,Y 369.298,Z 242.487,A -85,B 0,C 180,E1 -12867.819,E2 -12867.819} C_VEL
LIN {X 0,Y 369.208,Z 242.493,A -85,B 0,C 180,E1 -12871.091,E2 -12871.091} C_VEL
LIN {X 0,Y 369.307,Z 242.481,A -85,B 0,C 180,E1 -12872.181,E2 -12872.181} C_VEL
LIN {X 0,Y 368.983,Z 242.727,A -85,B 0,C 180,E1 -12875.191,E2 -12875.191} C_VEL
LIN {X 0,Y 368.761,Z 249.783,A -85,B 0,C 180,E1 -12878.77,E2 -12878.77} C_VEL
LIN {X 0,Y 368.626,Z 257.418,A -85,B 0,C 180,E1 -12882.665,E2 -12882.665} C_VEL
LIN {X 0,Y 368.419,Z 264.085,A -85,B 0,C 180,E1 -12886.058,E2 -12886.058} C_VEL
LIN {X 0,Y 368.295,Z 269.698,A -85,B 0,C 180,E1 -12888.929,E2 -12888.929} C_VEL
LIN {X 0,Y 368.215,Z 275.878,A -85,B 0,C 180,E1 -12891.998,E2 -12891.998} C_VEL
LIN {X 0,Y 370.072,Z 285.731,A -85,B 0,C 180,E1 -12892.469,E2 -12892.469} C_VEL
LIN {X 0,Y 371.572,Z 295.796,A -85,B 0,C 180,E1 -12893.108,E2 -12893.108} C_VEL
LIN {X 0,Y 371.114,Z 305.8,A -85,B 0,C 180,E1 -12893.878,E2 -12893.878} C_VEL
LIN {X 0,Y 370.557,Z 315.051,A -85,B 0,C 180,E1 -12894.811,E2 -12894.811} C_VEL
LIN {X 0,Y 370.05,Z 322.6,A -85,B 0,C 180,E1 -12895.75,E2 -12895.75} C_VEL
LIN {X 0,Y 369.489,Z 329.958,A -85,B 0,C 180,E1 -12896.865,E2 -12896.865} C_VEL
LIN {X 0,Y 368.936,Z 336.756,A -85,B 0,C 180,E1 -12898.13,E2 -12898.13} C_VEL
LIN {X 0,Y 368.433,Z 343.443,A -85,B 0,C 180,E1 -12899.733,E2 -12899.733} C_VEL
LIN {X 0,Y 368.088,Z 347.947,A -85,B 0,C 180,E1 -12901.139,E2 -12901.139} C_VEL
LIN {X 0,Y 367.229,Z 350.265,A -85,B 0,C 180,E1 -12901.983,E2 -12901.983} C_VEL
LIN {X 0,Y 364.111,Z 353.274,A -85,B 0,C 180,E1 -12903.382,E2 -12903.382} C_VEL
LIN {X 0,Y 361.078,Z 355.423,A -85,B 0,C 180,E1 -12904.838,E2 -12904.838} C_VEL
LIN {X 0,Y 360.364,Z 356.253,A -85,B 0,C 180,E1 -12905.76,E2 -12905.76} C_VEL
LIN {X 0,Y 360.341,Z 356.812,A -85,B 0,C 180,E1 -12907.201,E2 -12907.201} C_VEL
LIN {X 0,Y 360.411,Z 356.489,A -85,B 0,C 180,E1 -12908.739,E2 -12908.739} C_VEL
LIN {X 0,Y 360.62,Z 354.835,A -85,B 0,C 180,E1 -12910.53,E2 -12910.53} C_VEL
LIN {X 0,Y 360.813,Z 353.513,A -85,B 0,C 180,E1 -12911.473,E2 -12911.473} C_VEL
LIN {X 0,Y 361.157,Z 350.596,A -85,B 0,C 180,E1 -12912.929,E2 -12912.929} C_VEL
LIN {X 0,Y 361.547,Z 346.534,A -85,B 0,C 180,E1 -12914.411,E2 -12914.411} C_VEL
LIN {X 0,Y 361.996,Z 342.191,A -85,B 0,C 180,E1 -12915.659,E2 -12915.659} C_VEL
LIN {X 0,Y 362.6,Z 336.592,A -85,B 0,C 180,E1 -12916.952,E2 -12916.952} C_VEL
LIN {X 0,Y 363.184,Z 330.176,A -85,B 0,C 180,E1 -12918.161,E2 -12918.161} C_VEL
LIN {X 0,Y 363.935,Z 322.841,A -85,B 0,C 180,E1 -12919.284,E2 -12919.284} C_VEL
LIN {X 0,Y 364.719,Z 313.619,A -85,B 0,C 180,E1 -12920.425,E2 -12920.425} C_VEL
LIN {X 0,Y 365.344,Z 304.379,A -85,B 0,C 180,E1 -12921.303,E2 -12921.303} C_VEL
LIN {X 0,Y 365.597,Z 297.256,A -85,B 0,C 180,E1 -12921.862,E2 -12921.862} C_VEL
LIN {X 0,Y 363.873,Z 287.273,A -85,B 0,C 180,E1 -12922.564,E2 -12922.564} C_VEL
LIN {X 0,Y 361.666,Z 277.986,A -85,B 0,C 180,E1 -12923.088,E2 -12923.088} C_VEL
LIN {X 0,Y 361.471,Z 276.9,A -85,B 0,C 180,E1 -12923.152,E2 -12923.152} C_VEL
LIN {X 0,Y 361.635,Z 270.015,A -85,B 0,C 180,E1 -12926.685,E2 -12926.685} C_VEL
LIN {X 0,Y 361.869,Z 262.927,A -85,B 0,C 180,E1 -12930.314,E2 -12930.314} C_VEL
LIN {X 0,Y 361.981,Z 256.665,A -85,B 0,C 180,E1 -12933.477,E2 -12933.477} C_VEL
LIN {X 0,Y 362.21,Z 250.59,A -85,B 0,C 180,E1 -12936.561,E2 -12936.561} C_VEL
LIN {X 0,Y 362.255,Z 246.355,A -85,B 0,C 180,E1 -12938.628,E2 -12938.628} C_VEL
LIN {X 0,Y 361.894,Z 243.408,A -85,B 0,C 180,E1 -12940.132,E2 -12940.132} C_VEL
LIN {X 0,Y 361.935,Z 243.403,A -85,B 0,C 180,E1 -12943.066,E2 -12943.066} C_VEL
LIN {X 0,Y 362.001,Z 243.394,A -85,B 0,C 180,E1 -12946.528,E2 -12946.528} C_VEL
LIN {X 0,Y 362.034,Z 243.391,A -85,B 0,C 180,E1 -12949.938,E2 -12949.938} C_VEL
LIN {X 0,Y 362.128,Z 243.379,A -85,B 0,C 180,E1 -12953.313,E2 -12953.313} C_VEL
LIN {X 0,Y 362.283,Z 243.359,A -85,B 0,C 180,E1 -12957.776,E2 -12957.776} C_VEL
LIN {X 0,Y 362.429,Z 243.34,A -85,B 0,C 180,E1 -12960,E2 -12960} C_VEL
LIN {X 0,Y 362.283,Z 243.359,A -85,B 0,C 180,E1 -12962.223,E2 -12962.223} C_VEL
LIN {X 0,Y 362.138,Z 243.376,A -85,B 0,C 180,E1 -12966.687,E2 -12966.687} C_VEL
LIN {X 0,Y 362.033,Z 243.39,A -85,B 0,C 180,E1 -12970.062,E2 -12970.062} C_VEL
LIN {X 0,Y 362,Z 243.391,A -85,B 0,C 180,E1 -12973.899,E2 -12973.899} C_VEL
LIN {X 0,Y 361.969,Z 243.397,A -85,B 0,C 180,E1 -12977.938,E2 -12977.938} C_VEL
LIN {X 0,Y 361.862,Z 243.409,A -85,B 0,C 180,E1 -12981.655,E2 -12981.655} C_VEL
LIN {X 0,Y 361.927,Z 243.404,A -85,B 0,C 180,E1 -12985.29,E2 -12985.29} C_VEL
LIN {X 0,Y 361.92,Z 243.404,A -85,B 0,C 180,E1 -12987.778,E2 -12987.778} C_VEL
LIN {X 0,Y 361.848,Z 243.412,A -85,B 0,C 180,E1 -12991.285,E2 -12991.285} C_VEL
LIN {X 0,Y 361.855,Z 243.41,A -85,B 0,C 180,E1 -12994.28,E2 -12994.28} C_VEL
LIN {X 0,Y 361.865,Z 243.408,A -85,B 0,C 180,E1 -12997.223,E2 -12997.223} C_VEL
LIN {X 0,Y 361.837,Z 243.415,A -85,B 0,C 180,E1 -13000.756,E2 -13000.756} C_VEL
LIN {X 0,Y 361.818,Z 243.417,A -85,B 0,C 180,E1 -13004.368,E2 -13004.368} C_VEL
LIN {X 0,Y 361.895,Z 243.493,A -85,B 0,C 180,E1 -13006.134,E2 -13006.134} C_VEL
LIN {X 0,Y 362.948,Z 249.473,A -85,B 0,C 180,E1 -13009.694,E2 -13009.694} C_VEL
LIN {X 0,Y 363.758,Z 254.2,A -85,B 0,C 180,E1 -13012.386,E2 -13012.386} C_VEL
LIN {X 0,Y 363.892,Z 258.245,A -85,B 0,C 180,E1 -13014.591,E2 -13014.591} C_VEL
LIN {X 0,Y 363.355,Z 263.275,A -85,B 0,C 180,E1 -13017.209,E2 -13017.209} C_VEL
LIN {X 0,Y 362.496,Z 270.759,A -85,B 0,C 180,E1 -13021.007,E2 -13021.007} C_VEL
LIN {X 0,Y 361.848,Z 278.191,A -85,B 0,C 180,E1 -13024.704,E2 -13024.704} C_VEL
LIN {X 0,Y 361.273,Z 285.557,A -85,B 0,C 180,E1 -13028.308,E2 -13028.308} C_VEL
LIN {X 0,Y 360.927,Z 291.516,A -85,B 0,C 180,E1 -13031.186,E2 -13031.186} C_VEL
LIN {X 0,Y 362.726,Z 306.93,A -85,B 0,C 180,E1 -13031.94,E2 -13031.94} C_VEL
LIN {X 0,Y 364.105,Z 319.525,A -85,B 0,C 180,E1 -13032.76,E2 -13032.76} C_VEL
LIN {X 0,Y 364.703,Z 326.997,A -85,B 0,C 180,E1 -13033.343,E2 -13033.343} C_VEL
LIN {X 0,Y 363.778,Z 339.1,A -85,B 0,C 180,E1 -13034.451,E2 -13034.451} C_VEL
LIN {X 0,Y 362.888,Z 349.527,A -85,B 0,C 180,E1 -13035.636,E2 -13035.636} C_VEL
LIN {X 0,Y 362.267,Z 358.146,A -85,B 0,C 180,E1 -13036.824,E2 -13036.824} C_VEL
LIN {X 0,Y 361.64,Z 366.631,A -85,B 0,C 180,E1 -13038.226,E2 -13038.226} C_VEL
LIN {X 0,Y 361.077,Z 374.92,A -85,B 0,C 180,E1 -13039.911,E2 -13039.911} C_VEL
LIN {X 0,Y 360.753,Z 381.615,A -85,B 0,C 180,E1 -13041.598,E2 -13041.598} C_VEL
LIN {X 0,Y 360.569,Z 386.937,A -85,B 0,C 180,E1 -13043.284,E2 -13043.284} C_VEL
LIN {X 0,Y 360.543,Z 391.037,A -85,B 0,C 180,E1 -13044.968,E2 -13044.968} C_VEL
LIN {X 0,Y 360.447,Z 394.009,A -85,B 0,C 180,E1 -13046.647,E2 -13046.647} C_VEL
LIN {X 0,Y 360.585,Z 395.434,A -85,B 0,C 180,E1 -13047.766,E2 -13047.766} C_VEL
LIN {X 0,Y 360.541,Z 396.389,A -85,B 0,C 180,E1 -13048.883,E2 -13048.883} C_VEL
LIN {X 0,Y 360.521,Z 396.931,A -85,B 0,C 180,E1 -13050,E2 -13050} C_VEL
LIN {X 0,Y 360.521,Z 397.062,A -85,B 0,C 180,E1 -13051.117,E2 -13051.117} C_VEL
LIN {X 0,Y 360.443,Z 396.728,A -85,B 0,C 180,E1 -13052.235,E2 -13052.235} C_VEL
LIN {X 0,Y 360.387,Z 394.815,A -85,B 0,C 180,E1 -13054.474,E2 -13054.474} C_VEL
LIN {X 0,Y 360.385,Z 392.586,A -85,B 0,C 180,E1 -13055.972,E2 -13055.972} C_VEL
LIN {X 0,Y 360.644,Z 388.709,A -85,B 0,C 180,E1 -13057.84,E2 -13057.84} C_VEL
LIN {X 0,Y 360.992,Z 384.084,A -85,B 0,C 180,E1 -13059.526,E2 -13059.526} C_VEL
LIN {X 0,Y 361.725,Z 377.253,A -85,B 0,C 180,E1 -13061.487,E2 -13061.487} C_VEL
LIN {X 0,Y 362.995,Z 368.521,A -85,B 0,C 180,E1 -13063.435,E2 -13063.435} C_VEL
LIN {X 0,Y 364.002,Z 359.777,A -85,B 0,C 180,E1 -13065.034,E2 -13065.034} C_VEL
LIN {X 0,Y 365.702,Z 349.025,A -85,B 0,C 180,E1 -13066.611,E2 -13066.611} C_VEL
LIN {X 0,Y 367.382,Z 337.691,A -85,B 0,C 180,E1 -13067.967,E2 -13067.967} C_VEL
LIN {X 0,Y 368.356,Z 329.637,A -85,B 0,C 180,E1 -13068.782,E2 -13068.782} C_VEL
LIN {X 0,Y 368.224,Z 318.291,A -85,B 0,C 180,E1 -13069.869,E2 -13069.869} C_VEL
LIN {X 0,Y 366.674,Z 306.008,A -85,B 0,C 180,E1 -13070.973,E2 -13070.973} C_VEL
LIN {X 0,Y 363.783,Z 293.485,A -85,B 0,C 180,E1 -13072.059,E2 -13072.059} C_VEL
LIN {X 0,Y 361.711,Z 286.53,A -85,B 0,C 180,E1 -13072.653,E2 -13072.653} C_VEL
LIN {X 0,Y 361.619,Z 285.813,A -85,B 0,C 180,E1 -13072.751,E2 -13072.751} C_VEL
LIN {X 0,Y 362.349,Z 278.842,A -85,B 0,C 180,E1 -13076.494,E2 -13076.494} C_VEL
LIN {X 0,Y 363.25,Z 272.529,A -85,B 0,C 180,E1 -13080.202,E2 -13080.202} C_VEL
LIN {X 0,Y 364.351,Z 266.776,A -85,B 0,C 180,E1 -13084.014,E2 -13084.014} C_VEL
LIN {X 0,Y 364.841,Z 263.357,A -85,B 0,C 180,E1 -13086.667,E2 -13086.667} C_VEL
LIN {X 0,Y 364.779,Z 260.273,A -85,B 0,C 180,E1 -13089.587,E2 -13089.587} C_VEL
LIN {X 0,Y 364.37,Z 257.611,A -85,B 0,C 180,E1 -13092.866,E2 -13092.866} C_VEL
LIN {X 0,Y 364.071,Z 255.802,A -85,B 0,C 180,E1 -13095.977,E2 -13095.977} C_VEL
LIN {X 0,Y 363.823,Z 254.697,A -85,B 0,C 180,E1 -13098.945,E2 -13098.945} C_VEL
LIN {X 0,Y 363.623,Z 254.109,A -85,B 0,C 180,E1 -13102.414,E2 -13102.414} C_VEL
LIN {X 0,Y 363.522,Z 254.087,A -85,B 0,C 180,E1 -13104.55,E2 -13104.55} C_VEL
LIN {X 0,Y 363.156,Z 254.44,A -85,B 0,C 180,E1 -13107.189,E2 -13107.189} C_VEL
LIN {X 0,Y 362.657,Z 255.494,A -85,B 0,C 180,E1 -13111.022,E2 -13111.022} C_VEL
LIN {X 0,Y 362.215,Z 257.029,A -85,B 0,C 180,E1 -13114.731,E2 -13114.731} C_VEL
LIN {X 0,Y 361.893,Z 258.98,A -85,B 0,C 180,E1 -13118.458,E2 -13118.458} C_VEL
LIN {X 0,Y 363.074,Z 262.056,A -85,B 0,C 180,E1 -13118.804,E2 -13118.804} C_VEL
LIN {X 0,Y 367.338,Z 271.845,A -85,B 0,C 180,E1 -13119.933,E2 -13119.933} C_VEL
LIN {X 0,Y 370.506,Z 281.574,A -85,B 0,C 180,E1 -13121.027,E2 -13121.027} C_VEL
LIN {X 0,Y 371.599,Z 286.611,A -85,B 0,C 180,E1 -13121.583,E2 -13121.583} C_VEL
LIN {X 0,Y 370.092,Z 299.113,A -85,B 0,C 180,E1 -13122.74,E2 -13122.74} C_VEL
LIN {X 0,Y 368.425,Z 310.645,A -85,B 0,C 180,E1 -13124.085,E2 -13124.085} C_VEL
LIN {X 0,Y 367.085,Z 319.234,A -85,B 0,C 180,E1 -13125.305,E2 -13125.305} C_VEL
LIN {X 0,Y 365.815,Z 327.254,A -85,B 0,C 180,E1 -13126.671,E2 -13126.671} C_VEL
LIN {X 0,Y 364.472,Z 335.212,A -85,B 0,C 180,E1 -13128.319,E2 -13128.319} C_VEL
LIN {X 0,Y 363.34,Z 341.659,A -85,B 0,C 180,E1 -13129.975,E2 -13129.975} C_VEL
LIN {X 0,Y 362.435,Z 346.695,A -85,B 0,C 180,E1 -13131.582,E2 -13131.582} C_VEL
LIN {X 0,Y 361.911,Z 350.883,A -85,B 0,C 180,E1 -13133.309,E2 -13133.309} C_VEL
LIN {X 0,Y 361.599,Z 353.013,A -85,B 0,C 180,E1 -13134.423,E2 -13134.423} C_VEL
LIN {X 0,Y 361.327,Z 354.723,A -85,B 0,C 180,E1 -13135.538,E2 -13135.538} C_VEL
LIN {X 0,Y 361.213,Z 355.963,A -85,B 0,C 180,E1 -13136.654,E2 -13136.654} C_VEL
LIN {X 0,Y 360.821,Z 356.836,A -85,B 0,C 180,E1 -13137.768,E2 -13137.768} C_VEL
LIN {X 0,Y 360.644,Z 357.303,A -85,B 0,C 180,E1 -13138.884,E2 -13138.884} C_VEL
LIN {X 0,Y 360.558,Z 357.347,A -85,B 0,C 180,E1 -13140,E2 -13140} C_VEL
LIN {X 0,Y 360.56,Z 356.957,A -85,B 0,C 180,E1 -13141.117,E2 -13141.117} C_VEL
LIN {X 0,Y 360.601,Z 356.172,A -85,B 0,C 180,E1 -13142.234,E2 -13142.234} C_VEL
LIN {X 0,Y 360.566,Z 354.993,A -85,B 0,C 180,E1 -13143.352,E2 -13143.352} C_VEL
LIN {X 0,Y 360.688,Z 352.38,A -85,B 0,C 180,E1 -13145.03,E2 -13145.03} C_VEL
LIN {X 0,Y 360.864,Z 347.98,A -85,B 0,C 180,E1 -13147.002,E2 -13147.002} C_VEL
LIN {X 0,Y 361.196,Z 342.106,A -85,B 0,C 180,E1 -13148.955,E2 -13148.955} C_VEL
LIN {X 0,Y 361.657,Z 335.643,A -85,B 0,C 180,E1 -13150.639,E2 -13150.639} C_VEL
LIN {X 0,Y 362.268,Z 327.589,A -85,B 0,C 180,E1 -13152.322,E2 -13152.322} C_VEL
LIN {X 0,Y 363.057,Z 317.63,A -85,B 0,C 180,E1 -13154.003,E2 -13154.003} C_VEL
LIN {X 0,Y 363.775,Z 307.333,A -85,B 0,C 180,E1 -13155.405,E2 -13155.405} C_VEL
LIN {X 0,Y 364.621,Z 295.937,A -85,B 0,C 180,E1 -13156.661,E2 -13156.661} C_VEL
LIN {X 0,Y 365.437,Z 285.017,A -85,B 0,C 180,E1 -13157.632,E2 -13157.632} C_VEL
LIN {X 0,Y 365.74,Z 278.313,A -85,B 0,C 180,E1 -13158.13,E2 -13158.13} C_VEL
LIN {X 0,Y 363.145,Z 264.84,A -85,B 0,C 180,E1 -13159.045,E2 -13159.045} C_VEL
LIN {X 0,Y 360.717,Z 252.601,A -85,B 0,C 180,E1 -13159.676,E2 -13159.676} C_VEL
LIN {X 0,Y 360.736,Z 248.534,A -85,B 0,C 180,E1 -13163.697,E2 -13163.697} C_VEL
LIN {X 0,Y 360.859,Z 245.659,A -85,B 0,C 180,E1 -13166.612,E2 -13166.612} C_VEL
LIN {X 0,Y 360.911,Z 243.54,A -85,B 0,C 180,E1 -13168.802,E2 -13168.802} C_VEL
LIN {X 0,Y 361.439,Z 243.463,A -85,B 0,C 180,E1 -13172.987,E2 -13172.987} C_VEL
LIN {X 0,Y 361.722,Z 243.428,A -85,B 0,C 180,E1 -13175.654,E2 -13175.654} C_VEL
LIN {X 0,Y 361.866,Z 243.411,A -85,B 0,C 180,E1 -13179.025,E2 -13179.025} C_VEL
LIN {X 0,Y 361.839,Z 243.414,A -85,B 0,C 180,E1 -13182.829,E2 -13182.829} C_VEL
LIN {X 0,Y 361.82,Z 243.413,A -85,B 0,C 180,E1 -13185.947,E2 -13185.947} C_VEL
LIN {X 0,Y 361.815,Z 243.416,A -85,B 0,C 180,E1 -13189.249,E2 -13189.249} C_VEL
LIN {X 0,Y 361.864,Z 243.411,A -85,B 0,C 180,E1 -13192.981,E2 -13192.981} C_VEL
LIN {X 0,Y 361.861,Z 243.413,A -85,B 0,C 180,E1 -13196.631,E2 -13196.631} C_VEL
LIN {X 0,Y 361.87,Z 243.406,A -85,B 0,C 180,E1 -13199.671,E2 -13199.671} C_VEL
LIN {X 0,Y 361.904,Z 243.402,A -85,B 0,C 180,E1 -13203.471,E2 -13203.471} C_VEL
LIN {X 0,Y 361.882,Z 243.405,A -85,B 0,C 180,E1 -13207.144,E2 -13207.144} C_VEL
LIN {X 0,Y 361.91,Z 243.404,A -85,B 0,C 180,E1 -13210.723,E2 -13210.723} C_VEL
LIN {X 0,Y 361.936,Z 243.398,A -85,B 0,C 180,E1 -13213.066,E2 -13213.066} C_VEL
LIN {X 0,Y 362.003,Z 243.392,A -85,B 0,C 180,E1 -13216.528,E2 -13216.528} C_VEL
LIN {X 0,Y 362.003,Z 243.394,A -85,B 0,C 180,E1 -13219.937,E2 -13219.937} C_VEL
LIN {X 0,Y 362.12,Z 243.376,A -85,B 0,C 180,E1 -13223.313,E2 -13223.313} C_VEL
LIN {X 0,Y 362.26,Z 243.363,A -85,B 0,C 180,E1 -13227.776,E2 -13227.776} C_VEL
LIN {X 0,Y 362.179,Z 243.368,A -85,B 0,C 180,E1 -13231.112,E2 -13231.112} C_VEL
LIN {X 0,Y 362.269,Z 243.358,A -85,B 0,C 180,E1 -13232.223,E2 -13232.223} C_VEL
LIN {X 0,Y 361.912,Z 243.484,A -85,B 0,C 180,E1 -13235.013,E2 -13235.013} C_VEL
LIN {X 0,Y 361.791,Z 248.957,A -85,B 0,C 180,E1 -13237.815,E2 -13237.815} C_VEL
LIN {X 0,Y 361.606,Z 256.659,A -85,B 0,C 180,E1 -13241.775,E2 -13241.775} C_VEL
LIN {X 0,Y 361.423,Z 263.349,A -85,B 0,C 180,E1 -13245.219,E2 -13245.219} C_VEL
LIN {X 0,Y 361.285,Z 270.162,A -85,B 0,C 180,E1 -13248.722,E2 -13248.722} C_VEL
LIN {X 0,Y 361.164,Z 276.119,A -85,B 0,C 180,E1 -13251.736,E2 -13251.736} C_VEL
LIN {X 0,Y 363.013,Z 285.991,A -85,B 0,C 180,E1 -13252.218,E2 -13252.218} C_VEL
LIN {X 0,Y 364.622,Z 296.465,A -85,B 0,C 180,E1 -13252.899,E2 -13252.899} C_VEL
LIN {X 0,Y 364.091,Z 307.182,A -85,B 0,C 180,E1 -13253.763,E2 -13253.763} C_VEL
LIN {X 0,Y 363.539,Z 316.019,A -85,B 0,C 180,E1 -13254.685,E2 -13254.685} C_VEL
LIN {X 0,Y 363.005,Z 323.675,A -85,B 0,C 180,E1 -13255.67,E2 -13255.67} C_VEL
LIN {X 0,Y 362.421,Z 331.298,A -85,B 0,C 180,E1 -13256.87,E2 -13256.87} C_VEL
LIN {X 0,Y 361.767,Z 338.885,A -85,B 0,C 180,E1 -13258.384,E2 -13258.384} C_VEL
LIN {X 0,Y 361.36,Z 344.162,A -85,B 0,C 180,E1 -13259.732,E2 -13259.732} C_VEL
LIN {X 0,Y 361.014,Z 348.354,A -85,B 0,C 180,E1 -13261.074,E2 -13261.074} C_VEL
LIN {X 0,Y 360.77,Z 351.566,A -85,B 0,C 180,E1 -13262.392,E2 -13262.392} C_VEL
LIN {X 0,Y 360.544,Z 354.018,A -85,B 0,C 180,E1 -13263.748,E2 -13263.748} C_VEL
LIN {X 0,Y 360.418,Z 355.598,A -85,B 0,C 180,E1 -13265.016,E2 -13265.016} C_VEL
LIN {X 0,Y 360.364,Z 356.253,A -85,B 0,C 180,E1 -13265.76,E2 -13265.76} C_VEL
LIN {X 0,Y 359.671,Z 356.838,A -85,B 0,C 180,E1 -13266.688,E2 -13266.688} C_VEL
LIN {X 0,Y 358.079,Z 356.996,A -85,B 0,C 180,E1 -13267.601,E2 -13267.601} C_VEL
LIN {X 0,Y 355.551,Z 356.743,A -85,B 0,C 180,E1 -13268.814,E2 -13268.814} C_VEL
LIN {X 0,Y 353.751,Z 355.898,A -85,B 0,C 180,E1 -13270.057,E2 -13270.057} C_VEL
LIN {X 0,Y 353.562,Z 355.082,A -85,B 0,C 180,E1 -13270.69,E2 -13270.69} C_VEL
LIN {X 0,Y 353.792,Z 353.7,A -85,B 0,C 180,E1 -13271.718,E2 -13271.718} C_VEL
LIN {X 0,Y 354.179,Z 350.441,A -85,B 0,C 180,E1 -13273.301,E2 -13273.301} C_VEL
LIN {X 0,Y 354.65,Z 345.868,A -85,B 0,C 180,E1 -13274.926,E2 -13274.926} C_VEL
LIN {X 0,Y 355.145,Z 341.434,A -85,B 0,C 180,E1 -13276.162,E2 -13276.162} C_VEL
LIN {X 0,Y 355.759,Z 335.909,A -85,B 0,C 180,E1 -13277.417,E2 -13277.417} C_VEL
LIN {X 0,Y 356.534,Z 328.548,A -85,B 0,C 180,E1 -13278.774,E2 -13278.774} C_VEL
LIN {X 0,Y 357.418,Z 319.491,A -85,B 0,C 180,E1 -13280.073,E2 -13280.073} C_VEL
LIN {X 0,Y 358.085,Z 311.425,A -85,B 0,C 180,E1 -13280.994,E2 -13280.994} C_VEL
LIN {X 0,Y 358.699,Z 303.036,A -85,B 0,C 180,E1 -13281.765,E2 -13281.765} C_VEL
LIN {X 0,Y 358.826,Z 298.614,A -85,B 0,C 180,E1 -13282.127,E2 -13282.127} C_VEL
LIN {X 0,Y 357.018,Z 288.061,A -85,B 0,C 180,E1 -13282.897,E2 -13282.897} C_VEL
LIN {X 0,Y 354.759,Z 278.646,A -85,B 0,C 180,E1 -13283.449,E2 -13283.449} C_VEL
LIN {X 0,Y 354.49,Z 277.238,A -85,B 0,C 180,E1 -13283.534,E2 -13283.534} C_VEL
LIN {X 0,Y 354.646,Z 270.571,A -85,B 0,C 180,E1 -13287.003,E2 -13287.003} C_VEL
LIN {X 0,Y 354.885,Z 263.572,A -85,B 0,C 180,E1 -13290.617,E2 -13290.617} C_VEL
LIN {X 0,Y 355.009,Z 257.853,A -85,B 0,C 180,E1 -13293.584,E2 -13293.584} C_VEL
LIN {X 0,Y 355.224,Z 251.657,A -85,B 0,C 180,E1 -13296.691,E2 -13296.691} C_VEL
LIN {X 0,Y 355.218,Z 246.833,A -85,B 0,C 180,E1 -13299.137,E2 -13299.137} C_VEL
LIN {X 0,Y 354.842,Z 244.287,A -85,B 0,C 180,E1 -13300.474,E2 -13300.474} C_VEL
LIN {X 0,Y 354.892,Z 244.28,A -85,B 0,C 180,E1 -13303.904,E2 -13303.904} C_VEL
LIN {X 0,Y 354.924,Z 244.276,A -85,B 0,C 180,E1 -13307.419,E2 -13307.419} C_VEL
LIN {X 0,Y 355.002,Z 244.267,A -85,B 0,C 180,E1 -13310.887,E2 -13310.887} C_VEL
LIN {X 0,Y 355.074,Z 244.257,A -85,B 0,C 180,E1 -13314.32,E2 -13314.32} C_VEL
LIN {X 0,Y 355.246,Z 244.235,A -85,B 0,C 180,E1 -13317.732,E2 -13317.732} C_VEL
LIN {X 0,Y 355.398,Z 244.216,A -85,B 0,C 180,E1 -13320,E2 -13320} C_VEL
LIN {X 0,Y 355.246,Z 244.235,A -85,B 0,C 180,E1 -13322.267,E2 -13322.267} C_VEL
LIN {X 0,Y 355.102,Z 244.253,A -85,B 0,C 180,E1 -13326.82,E2 -13326.82} C_VEL
LIN {X 0,Y 354.98,Z 244.268,A -85,B 0,C 180,E1 -13330.264,E2 -13330.264} C_VEL
LIN {X 0,Y 354.945,Z 244.27,A -85,B 0,C 180,E1 -13334.019,E2 -13334.019} C_VEL
LIN {X 0,Y 354.924,Z 244.274,A -85,B 0,C 180,E1 -13338.108,E2 -13338.108} C_VEL
LIN {X 0,Y 354.817,Z 244.288,A -85,B 0,C 180,E1 -13342.107,E2 -13342.107} C_VEL
LIN {X 0,Y 354.899,Z 244.279,A -85,B 0,C 180,E1 -13345.827,E2 -13345.827} C_VEL
LIN {X 0,Y 354.855,Z 244.281,A -85,B 0,C 180,E1 -13349.678,E2 -13349.678} C_VEL
LIN {X 0,Y 354.807,Z 244.289,A -85,B 0,C 180,E1 -13353.702,E2 -13353.702} C_VEL
LIN {X 0,Y 354.799,Z 244.29,A -85,B 0,C 180,E1 -13356.459,E2 -13356.459} C_VEL
LIN {X 0,Y 354.825,Z 244.285,A -85,B 0,C 180,E1 -13359.424,E2 -13359.424} C_VEL
LIN {X 0,Y 354.789,Z 244.292,A -85,B 0,C 180,E1 -13362.867,E2 -13362.867} C_VEL
LIN {X 0,Y 354.845,Z 244.344,A -85,B 0,C 180,E1 -13365.915,E2 -13365.915} C_VEL
LIN {X 0,Y 355.83,Z 249.942,A -85,B 0,C 180,E1 -13369.324,E2 -13369.324} C_VEL
LIN {X 0,Y 356.719,Z 255.141,A -85,B 0,C 180,E1 -13372.356,E2 -13372.356} C_VEL
LIN {X 0,Y 356.862,Z 259.015,A -85,B 0,C 180,E1 -13374.503,E2 -13374.503} C_VEL
LIN {X 0,Y 356.134,Z 265.233,A -85,B 0,C 180,E1 -13377.804,E2 -13377.804} C_VEL
LIN {X 0,Y 355.296,Z 272.681,A -85,B 0,C 180,E1 -13381.658,E2 -13381.658} C_VEL
LIN {X 0,Y 354.632,Z 280.062,A -85,B 0,C 180,E1 -13385.407,E2 -13385.407} C_VEL
LIN {X 0,Y 354.053,Z 288.626,A -85,B 0,C 180,E1 -13389.673,E2 -13389.673} C_VEL
LIN {X 0,Y 353.863,Z 291.438,A -85,B 0,C 180,E1 -13390.984,E2 -13390.984} C_VEL
LIN {X 0,Y 355.443,Z 305.207,A -85,B 0,C 180,E1 -13391.638,E2 -13391.638} C_VEL
LIN {X 0,Y 356.863,Z 317.878,A -85,B 0,C 180,E1 -13392.461,E2 -13392.461} C_VEL
LIN {X 0,Y 357.625,Z 326.606,A -85,B 0,C 180,E1 -13393.15,E2 -13393.15} C_VEL
LIN {X 0,Y 356.768,Z 338.695,A -85,B 0,C 180,E1 -13394.285,E2 -13394.285} C_VEL
LIN {X 0,Y 355.835,Z 349.252,A -85,B 0,C 180,E1 -13395.511,E2 -13395.511} C_VEL
LIN {X 0,Y 355.123,Z 358.632,A -85,B 0,C 180,E1 -13396.845,E2 -13396.845} C_VEL
LIN {X 0,Y 354.369,Z 368.41,A -85,B 0,C 180,E1 -13398.561,E2 -13398.561} C_VEL
LIN {X 0,Y 353.897,Z 376.32,A -85,B 0,C 180,E1 -13400.282,E2 -13400.282} C_VEL
LIN {X 0,Y 353.606,Z 382.782,A -85,B 0,C 180,E1 -13402.003,E2 -13402.003} C_VEL
LIN {X 0,Y 353.405,Z 388.37,A -85,B 0,C 180,E1 -13403.895,E2 -13403.895} C_VEL
LIN {X 0,Y 353.429,Z 391.622,A -85,B 0,C 180,E1 -13405.438,E2 -13405.438} C_VEL
LIN {X 0,Y 353.501,Z 394.852,A -85,B 0,C 180,E1 -13407.721,E2 -13407.721} C_VEL
LIN {X 0,Y 353.478,Z 395.857,A -85,B 0,C 180,E1 -13408.861,E2 -13408.861} C_VEL
LIN {X 0,Y 353.456,Z 396.438,A -85,B 0,C 180,E1 -13410,E2 -13410} C_VEL
LIN {X 0,Y 353.455,Z 396.61,A -85,B 0,C 180,E1 -13411.14,E2 -13411.14} C_VEL
LIN {X 0,Y 353.344,Z 396.354,A -85,B 0,C 180,E1 -13412.28,E2 -13412.28} C_VEL
LIN {X 0,Y 353.278,Z 395.643,A -85,B 0,C 180,E1 -13413.422,E2 -13413.422} C_VEL
LIN {X 0,Y 353.298,Z 394.527,A -85,B 0,C 180,E1 -13414.564,E2 -13414.564} C_VEL
LIN {X 0,Y 353.296,Z 392.653,A -85,B 0,C 180,E1 -13415.937,E2 -13415.937} C_VEL
LIN {X 0,Y 353.568,Z 388.603,A -85,B 0,C 180,E1 -13417.998,E2 -13417.998} C_VEL
LIN {X 0,Y 353.966,Z 384.091,A -85,B 0,C 180,E1 -13419.716,E2 -13419.716} C_VEL
LIN {X 0,Y 354.769,Z 377.395,A -85,B 0,C 180,E1 -13421.716,E2 -13421.716} C_VEL
LIN {X 0,Y 355.922,Z 370.233,A -85,B 0,C 180,E1 -13423.416,E2 -13423.416} C_VEL
LIN {X 0,Y 356.954,Z 361.85,A -85,B 0,C 180,E1 -13425.063,E2 -13425.063} C_VEL
LIN {X 0,Y 358.763,Z 350.919,A -85,B 0,C 180,E1 -13426.795,E2 -13426.795} C_VEL
LIN {X 0,Y 360.509,Z 340.11,A -85,B 0,C 180,E1 -13428.175,E2 -13428.175} C_VEL
LIN {X 0,Y 361.815,Z 331.208,A -85,B 0,C 180,E1 -13429.135,E2 -13429.135} C_VEL
LIN {X 0,Y 361.862,Z 320.38,A -85,B 0,C 180,E1 -13430.233,E2 -13430.233} C_VEL
LIN {X 0,Y 360.444,Z 307.87,A -85,B 0,C 180,E1 -13431.438,E2 -13431.438} C_VEL
LIN {X 0,Y 358.063,Z 296.785,A -85,B 0,C 180,E1 -13432.478,E2 -13432.478} C_VEL
LIN {X 0,Y 355.446,Z 288.27,A -85,B 0,C 180,E1 -13433.294,E2 -13433.294} C_VEL
LIN {X 0,Y 354.743,Z 285.208,A -85,B 0,C 180,E1 -13433.565,E2 -13433.565} C_VEL
LIN {X 0,Y 355.455,Z 278.786,A -85,B 0,C 180,E1 -13437.16,E2 -13437.16} C_VEL
LIN {X 0,Y 356.419,Z 272.786,A -85,B 0,C 180,E1 -13440.843,E2 -13440.843} C_VEL
LIN {X 0,Y 357.426,Z 267.753,A -85,B 0,C 180,E1 -13444.326,E2 -13444.326} C_VEL
LIN {X 0,Y 357.866,Z 265.158,A -85,B 0,C 180,E1 -13446.372,E2 -13446.372} C_VEL
LIN {X 0,Y 357.87,Z 262.411,A -85,B 0,C 180,E1 -13448.935,E2 -13448.935} C_VEL
LIN {X 0,Y 357.535,Z 259.849,A -85,B 0,C 180,E1 -13451.939,E2 -13451.939} C_VEL
LIN {X 0,Y 357.214,Z 257.83,A -85,B 0,C 180,E1 -13455.096,E2 -13455.096} C_VEL
LIN {X 0,Y 356.916,Z 256.419,A -85,B 0,C 180,E1 -13458.44,E2 -13458.44} C_VEL
LIN {X 0,Y 356.701,Z 255.667,A -85,B 0,C 180,E1 -13462.01,E2 -13462.01} C_VEL
LIN {X 0,Y 356.495,Z 255.615,A -85,B 0,C 180,E1 -13465.13,E2 -13465.13} C_VEL
LIN {X 0,Y 356.058,Z 256.067,A -85,B 0,C 180,E1 -13468.077,E2 -13468.077} C_VEL
LIN {X 0,Y 355.776,Z 256.668,A -85,B 0,C 180,E1 -13470.406,E2 -13470.406} C_VEL
LIN {X 0,Y 355.29,Z 258.094,A -85,B 0,C 180,E1 -13474.203,E2 -13474.203} C_VEL
LIN {X 0,Y 354.94,Z 259.751,A -85,B 0,C 180,E1 -13477.633,E2 -13477.633} C_VEL
LIN {X 0,Y 356.029,Z 262.671,A -85,B 0,C 180,E1 -13477.955,E2 -13477.955} C_VEL
LIN {X 0,Y 358.102,Z 266.699,A -85,B 0,C 180,E1 -13478.485,E2 -13478.485} C_VEL
LIN {X 0,Y 362.579,Z 278.012,A -85,B 0,C 180,E1 -13479.875,E2 -13479.875} C_VEL
LIN {X 0,Y 365.212,Z 287.717,A -85,B 0,C 180,E1 -13481.04,E2 -13481.04} C_VEL
LIN {X 0,Y 365.197,Z 289.86,A -85,B 0,C 180,E1 -13481.248,E2 -13481.248} C_VEL
LIN {X 0,Y 363.567,Z 301.666,A -85,B 0,C 180,E1 -13482.42,E2 -13482.42} C_VEL
LIN {X 0,Y 361.814,Z 312.798,A -85,B 0,C 180,E1 -13483.786,E2 -13483.786} C_VEL
LIN {X 0,Y 360.129,Z 322.721,A -85,B 0,C 180,E1 -13485.304,E2 -13485.304} C_VEL
LIN {X 0,Y 358.554,Z 331.587,A -85,B 0,C 180,E1 -13486.973,E2 -13486.973} C_VEL
LIN {X 0,Y 357.197,Z 338.805,A -85,B 0,C 180,E1 -13488.653,E2 -13488.653} C_VEL
LIN {X 0,Y 356.199,Z 344.611,A -85,B 0,C 180,E1 -13490.345,E2 -13490.345} C_VEL
LIN {X 0,Y 355.133,Z 349.289,A -85,B 0,C 180,E1 -13492.037,E2 -13492.037} C_VEL
LIN {X 0,Y 354.741,Z 352.828,A -85,B 0,C 180,E1 -13493.745,E2 -13493.745} C_VEL
LIN {X 0,Y 354.29,Z 355.414,A -85,B 0,C 180,E1 -13495.449,E2 -13495.449} C_VEL
LIN {X 0,Y 354.162,Z 356.591,A -85,B 0,C 180,E1 -13496.587,E2 -13496.587} C_VEL
LIN {X 0,Y 353.761,Z 357.405,A -85,B 0,C 180,E1 -13497.723,E2 -13497.723} C_VEL
LIN {X 0,Y 353.578,Z 357.801,A -85,B 0,C 180,E1 -13498.861,E2 -13498.861} C_VEL
LIN {X 0,Y 353.492,Z 357.753,A -85,B 0,C 180,E1 -13500,E2 -13500} C_VEL
LIN {X 0,Y 353.496,Z 357.306,A -85,B 0,C 180,E1 -13501.139,E2 -13501.139} C_VEL
LIN {X 0,Y 353.506,Z 356.467,A -85,B 0,C 180,E1 -13502.279,E2 -13502.279} C_VEL
LIN {X 0,Y 353.476,Z 355.199,A -85,B 0,C 180,E1 -13503.42,E2 -13503.42} C_VEL
LIN {X 0,Y 353.61,Z 352.484,A -85,B 0,C 180,E1 -13505.131,E2 -13505.131} C_VEL
LIN {X 0,Y 353.786,Z 348.269,A -85,B 0,C 180,E1 -13507.02,E2 -13507.02} C_VEL
LIN {X 0,Y 354.167,Z 341.935,A -85,B 0,C 180,E1 -13509.135,E2 -13509.135} C_VEL
LIN {X 0,Y 354.651,Z 335.302,A -85,B 0,C 180,E1 -13510.851,E2 -13510.851} C_VEL
LIN {X 0,Y 355.275,Z 327.073,A -85,B 0,C 180,E1 -13512.568,E2 -13512.568} C_VEL
LIN {X 0,Y 355.943,Z 318.83,A -85,B 0,C 180,E1 -13513.983,E2 -13513.983} C_VEL
LIN {X 0,Y 356.673,Z 308.656,A -85,B 0,C 180,E1 -13515.426,E2 -13515.426} C_VEL
LIN {X 0,Y 357.561,Z 297.448,A -85,B 0,C 180,E1 -13516.706,E2 -13516.706} C_VEL
LIN {X 0,Y 358.479,Z 285.089,A -85,B 0,C 180,E1 -13517.838,E2 -13517.838} C_VEL
LIN {X 0,Y 358.76,Z 279.483,A -85,B 0,C 180,E1 -13518.267,E2 -13518.267} C_VEL
LIN {X 0,Y 356.073,Z 265.37,A -85,B 0,C 180,E1 -13519.255,E2 -13519.255} C_VEL
LIN {X 0,Y 353.652,Z 252.933,A -85,B 0,C 180,E1 -13519.934,E2 -13519.934} C_VEL
LIN {X 0,Y 353.662,Z 248.943,A -85,B 0,C 180,E1 -13523.918,E2 -13523.918} C_VEL
LIN {X 0,Y 353.793,Z 245.758,A -85,B 0,C 180,E1 -13527.187,E2 -13527.187} C_VEL
LIN {X 0,Y 353.835,Z 244.526,A -85,B 0,C 180,E1 -13528.47,E2 -13528.47} C_VEL
LIN {X 0,Y 354.265,Z 244.354,A -85,B 0,C 180,E1 -13532.387,E2 -13532.387} C_VEL
LIN {X 0,Y 354.688,Z 244.304,A -85,B 0,C 180,E1 -13535.668,E2 -13535.668} C_VEL
LIN {X 0,Y 354.79,Z 244.289,A -85,B 0,C 180,E1 -13537.885,E2 -13537.885} C_VEL
LIN {X 0,Y 354.79,Z 244.293,A -85,B 0,C 180,E1 -13541.171,E2 -13541.171} C_VEL
LIN {X 0,Y 354.766,Z 244.293,A -85,B 0,C 180,E1 -13544.506,E2 -13544.506} C_VEL
LIN {X 0,Y 354.791,Z 244.288,A -85,B 0,C 180,E1 -13547.662,E2 -13547.662} C_VEL
LIN {X 0,Y 354.788,Z 244.292,A -85,B 0,C 180,E1 -13550.662,E2 -13550.662} C_VEL
LIN {X 0,Y 354.821,Z 244.286,A -85,B 0,C 180,E1 -13554.302,E2 -13554.302} C_VEL
LIN {X 0,Y 354.79,Z 244.288,A -85,B 0,C 180,E1 -13557.666,E2 -13557.666} C_VEL
LIN {X 0,Y 354.813,Z 244.285,A -85,B 0,C 180,E1 -13561.615,E2 -13561.615} C_VEL
LIN {X 0,Y 354.857,Z 244.28,A -85,B 0,C 180,E1 -13565.423,E2 -13565.423} C_VEL
LIN {X 0,Y 354.83,Z 244.284,A -85,B 0,C 180,E1 -13569.113,E2 -13569.113} C_VEL
LIN {X 0,Y 354.902,Z 244.276,A -85,B 0,C 180,E1 -13572.72,E2 -13572.72} C_VEL
LIN {X 0,Y 354.955,Z 244.273,A -85,B 0,C 180,E1 -13576.255,E2 -13576.255} C_VEL
LIN {X 0,Y 354.959,Z 244.27,A -85,B 0,C 180,E1 -13579.735,E2 -13579.735} C_VEL
LIN {X 0,Y 355.086,Z 244.252,A -85,B 0,C 180,E1 -13583.18,E2 -13583.18} C_VEL
LIN {X 0,Y 355.222,Z 244.239,A -85,B 0,C 180,E1 -13587.732,E2 -13587.732} C_VEL
LIN {X 0,Y 355.15,Z 244.244,A -85,B 0,C 180,E1 -13591.134,E2 -13591.134} C_VEL
LIN {X 0,Y 355.23,Z 244.234,A -85,B 0,C 180,E1 -13592.268,E2 -13592.268} C_VEL
LIN {X 0,Y 354.854,Z 244.378,A -85,B 0,C 180,E1 -13594.899,E2 -13594.899} C_VEL
LIN {X 0,Y 354.784,Z 249.472,A -85,B 0,C 180,E1 -13597.537,E2 -13597.537} C_VEL
LIN {X 0,Y 354.59,Z 256.993,A -85,B 0,C 180,E1 -13601.432,E2 -13601.432} C_VEL
LIN {X 0,Y 354.408,Z 263.768,A -85,B 0,C 180,E1 -13604.939,E2 -13604.939} C_VEL
LIN {X 0,Y 354.265,Z 270.6,A -85,B 0,C 180,E1 -13608.506,E2 -13608.506} C_VEL
LIN {X 0,Y 354.081,Z 276.308,A -85,B 0,C 180,E1 -13611.461,E2 -13611.461} C_VEL
LIN {X 0,Y 355.859,Z 285.808,A -85,B 0,C 180,E1 -13611.93,E2 -13611.93} C_VEL
LIN {X 0,Y 357.428,Z 295.202,A -85,B 0,C 180,E1 -13612.546,E2 -13612.546} C_VEL
LIN {X 0,Y 357.599,Z 299.232,A -85,B 0,C 180,E1 -13612.84,E2 -13612.84} C_VEL
LIN {X 0,Y 357.085,Z 308.547,A -85,B 0,C 180,E1 -13613.641,E2 -13613.641} C_VEL
LIN {X 0,Y 356.6,Z 316.101,A -85,B 0,C 180,E1 -13614.448,E2 -13614.448} C_VEL
LIN {X 0,Y 356.112,Z 322.442,A -85,B 0,C 180,E1 -13615.256,E2 -13615.256} C_VEL
LIN {X 0,Y 355.552,Z 329.895,A -85,B 0,C 180,E1 -13616.407,E2 -13616.407} C_VEL
LIN {X 0,Y 354.952,Z 336.87,A -85,B 0,C 180,E1 -13617.729,E2 -13617.729} C_VEL
LIN {X 0,Y 354.433,Z 343.274,A -85,B 0,C 180,E1 -13619.252,E2 -13619.252} C_VEL
LIN {X 0,Y 354.101,Z 347.114,A -85,B 0,C 180,E1 -13620.405,E2 -13620.405} C_VEL
LIN {X 0,Y 353.793,Z 350.954,A -85,B 0,C 180,E1 -13621.853,E2 -13621.853} C_VEL
LIN {X 0,Y 353.453,Z 354.558,A -85,B 0,C 180,E1 -13623.831,E2 -13623.831} C_VEL
LIN {X 0,Y 353.263,Z 356.5,A -85,B 0,C 180,E1 -13625.745,E2 -13625.745} C_VEL
LIN {X 0,Y 353.278,Z 357.205,A -85,B 0,C 180,E1 -13627.274,E2 -13627.274} C_VEL
LIN {X 0,Y 353.377,Z 356.339,A -85,B 0,C 180,E1 -13629.525,E2 -13629.525} C_VEL
LIN {X 0,Y 353.562,Z 355.082,A -85,B 0,C 180,E1 -13630.69,E2 -13630.69} C_VEL
LIN {X 0,Y 353.102,Z 353.919,A -85,B 0,C 180,E1 -13631.626,E2 -13631.626} C_VEL
LIN {X 0,Y 350.592,Z 351.305,A -85,B 0,C 180,E1 -13633.13,E2 -13633.13} C_VEL
LIN {X 0,Y 348.148,Z 347.839,A -85,B 0,C 180,E1 -13634.605,E2 -13634.605} C_VEL
LIN {X 0,Y 347.807,Z 345.159,A -85,B 0,C 180,E1 -13635.479,E2 -13635.479} C_VEL
LIN {X 0,Y 348.507,Z 339.547,A -85,B 0,C 180,E1 -13636.972,E2 -13636.972} C_VEL
LIN {X 0,Y 349.208,Z 332.752,A -85,B 0,C 180,E1 -13638.383,E2 -13638.383} C_VEL
LIN {X 0,Y 349.997,Z 325.899,A -85,B 0,C 180,E1 -13639.53,E2 -13639.53} C_VEL
LIN {X 0,Y 350.755,Z 317.886,A -85,B 0,C 180,E1 -13640.626,E2 -13640.626} C_VEL
LIN {X 0,Y 351.51,Z 309.064,A -85,B 0,C 180,E1 -13641.597,E2 -13641.597} C_VEL
LIN {X 0,Y 352.129,Z 300.773,A -85,B 0,C 180,E1 -13642.321,E2 -13642.321} C_VEL
LIN {X 0,Y 350.333,Z 289.603,A -85,B 0,C 180,E1 -13643.196,E2 -13643.196} C_VEL
LIN {X 0,Y 347.99,Z 279.629,A -85,B 0,C 180,E1 -13643.812,E2 -13643.812} C_VEL
LIN {X 0,Y 347.515,Z 277.627,A -85,B 0,C 180,E1 -13643.924,E2 -13643.924} C_VEL
LIN {X 0,Y 347.736,Z 269.679,A -85,B 0,C 180,E1 -13648.087,E2 -13648.087} C_VEL
LIN {X 0,Y 347.922,Z 262.845,A -85,B 0,C 180,E1 -13651.66,E2 -13651.66} C_VEL
LIN {X 0,Y 348.109,Z 256.57,A -85,B 0,C 180,E1 -13654.914,E2 -13654.914} C_VEL
LIN {X 0,Y 348.364,Z 250.333,A -85,B 0,C 180,E1 -13658.128,E2 -13658.128} C_VEL
LIN {X 0,Y 347.891,Z 245.662,A -85,B 0,C 180,E1 -13660.529,E2 -13660.529} C_VEL
LIN {X 0,Y 347.836,Z 245.159,A -85,B 0,C 180,E1 -13660.832,E2 -13660.832} C_VEL
LIN {X 0,Y 347.839,Z 245.157,A -85,B 0,C 180,E1 -13663.568,E2 -13663.568} C_VEL
LIN {X 0,Y 347.893,Z 245.151,A -85,B 0,C 180,E1 -13667.16,E2 -13667.16} C_VEL
LIN {X 0,Y 347.944,Z 245.147,A -85,B 0,C 180,E1 -13670.701,E2 -13670.701} C_VEL
LIN {X 0,Y 348.066,Z 245.131,A -85,B 0,C 180,E1 -13673.041,E2 -13673.041} C_VEL
LIN {X 0,Y 348.208,Z 245.111,A -85,B 0,C 180,E1 -13677.686,E2 -13677.686} C_VEL
LIN {X 0,Y 348.347,Z 245.094,A -85,B 0,C 180,E1 -13680,E2 -13680} C_VEL
LIN {X 0,Y 348.208,Z 245.112,A -85,B 0,C 180,E1 -13682.313,E2 -13682.313} C_VEL
LIN {X 0,Y 348.07,Z 245.129,A -85,B 0,C 180,E1 -13686.958,E2 -13686.958} C_VEL
LIN {X 0,Y 347.93,Z 245.146,A -85,B 0,C 180,E1 -13690.474,E2 -13690.474} C_VEL
LIN {X 0,Y 347.9,Z 245.148,A -85,B 0,C 180,E1 -13694.15,E2 -13694.15} C_VEL
LIN {X 0,Y 347.892,Z 245.149,A -85,B 0,C 180,E1 -13698.29,E2 -13698.29} C_VEL
LIN {X 0,Y 347.769,Z 245.164,A -85,B 0,C 180,E1 -13701.626,E2 -13701.626} C_VEL
LIN {X 0,Y 347.813,Z 245.161,A -85,B 0,C 180,E1 -13705.108,E2 -13705.108} C_VEL
LIN {X 0,Y 347.812,Z 245.162,A -85,B 0,C 180,E1 -13707.694,E2 -13707.694} C_VEL
LIN {X 0,Y 347.765,Z 245.166,A -85,B 0,C 180,E1 -13710.346,E2 -13710.346} C_VEL
LIN {X 0,Y 347.745,Z 245.167,A -85,B 0,C 180,E1 -13714.464,E2 -13714.464} C_VEL
LIN {X 0,Y 347.775,Z 245.165,A -85,B 0,C 180,E1 -13717.989,E2 -13717.989} C_VEL
LIN {X 0,Y 347.752,Z 245.166,A -85,B 0,C 180,E1 -13721.83,E2 -13721.83} C_VEL
LIN {X 0,Y 347.803,Z 245.239,A -85,B 0,C 180,E1 -13725.732,E2 -13725.732} C_VEL
LIN {X 0,Y 348.744,Z 250.622,A -85,B 0,C 180,E1 -13729.084,E2 -13729.084} C_VEL
LIN {X 0,Y 349.68,Z 256.013,A -85,B 0,C 180,E1 -13732.295,E2 -13732.295} C_VEL
LIN {X 0,Y 349.821,Z 259.655,A -85,B 0,C 180,E1 -13734.365,E2 -13734.365} C_VEL
LIN {X 0,Y 349.25,Z 264.664,A -85,B 0,C 180,E1 -13737.09,E2 -13737.09} C_VEL
LIN {X 0,Y 348.343,Z 272.095,A -85,B 0,C 180,E1 -13741.039,E2 -13741.039} C_VEL
LIN {X 0,Y 347.645,Z 279.458,A -85,B 0,C 180,E1 -13744.879,E2 -13744.879} C_VEL
LIN {X 0,Y 347.068,Z 286.867,A -85,B 0,C 180,E1 -13748.667,E2 -13748.667} C_VEL
LIN {X 0,Y 346.793,Z 290.923,A -85,B 0,C 180,E1 -13750.734,E2 -13750.734} C_VEL
LIN {X 0,Y 348.293,Z 304.594,A -85,B 0,C 180,E1 -13751.397,E2 -13751.397} C_VEL
LIN {X 0,Y 349.724,Z 317.548,A -85,B 0,C 180,E1 -13752.257,E2 -13752.257} C_VEL
LIN {X 0,Y 350.545,Z 327.777,A -85,B 0,C 180,E1 -13753.1,E2 -13753.1} C_VEL
LIN {X 0,Y 349.684,Z 339.576,A -85,B 0,C 180,E1 -13754.257,E2 -13754.257} C_VEL
LIN {X 0,Y 348.638,Z 350.06,A -85,B 0,C 180,E1 -13755.533,E2 -13755.533} C_VEL
LIN {X 0,Y 347.985,Z 359.031,A -85,B 0,C 180,E1 -13756.867,E2 -13756.867} C_VEL
LIN {X 0,Y 347.266,Z 368.678,A -85,B 0,C 180,E1 -13758.62,E2 -13758.62} C_VEL
LIN {X 0,Y 346.771,Z 376.998,A -85,B 0,C 180,E1 -13760.375,E2 -13760.375} C_VEL
LIN {X 0,Y 346.548,Z 382.502,A -85,B 0,C 180,E1 -13761.839,E2 -13761.839} C_VEL
LIN {X 0,Y 346.412,Z 386.074,A -85,B 0,C 180,E1 -13763.008,E2 -13763.008} C_VEL
LIN {X 0,Y 346.337,Z 389.001,A -85,B 0,C 180,E1 -13764.177,E2 -13764.177} C_VEL
LIN {X 0,Y 346.344,Z 391.302,A -85,B 0,C 180,E1 -13765.344,E2 -13765.344} C_VEL
LIN {X 0,Y 346.283,Z 393.008,A -85,B 0,C 180,E1 -13766.509,E2 -13766.509} C_VEL
LIN {X 0,Y 346.417,Z 395.318,A -85,B 0,C 180,E1 -13768.838,E2 -13768.838} C_VEL
LIN {X 0,Y 346.393,Z 395.941,A -85,B 0,C 180,E1 -13770,E2 -13770} C_VEL
LIN {X 0,Y 346.39,Z 396.155,A -85,B 0,C 180,E1 -13771.163,E2 -13771.163} C_VEL
LIN {X 0,Y 346.247,Z 395.949,A -85,B 0,C 180,E1 -13772.327,E2 -13772.327} C_VEL
LIN {X 0,Y 346.198,Z 395.319,A -85,B 0,C 180,E1 -13773.492,E2 -13773.492} C_VEL
LIN {X 0,Y 346.21,Z 394.247,A -85,B 0,C 180,E1 -13774.658,E2 -13774.658} C_VEL
LIN {X 0,Y 346.197,Z 392.683,A -85,B 0,C 180,E1 -13775.885,E2 -13775.885} C_VEL
LIN {X 0,Y 346.434,Z 389.739,A -85,B 0,C 180,E1 -13777.578,E2 -13777.578} C_VEL
LIN {X 0,Y 346.779,Z 385.704,A -85,B 0,C 180,E1 -13779.331,E2 -13779.331} C_VEL
LIN {X 0,Y 347.385,Z 380.571,A -85,B 0,C 180,E1 -13781.081,E2 -13781.081} C_VEL
LIN {X 0,Y 348.391,Z 374.248,A -85,B 0,C 180,E1 -13782.821,E2 -13782.821} C_VEL
LIN {X 0,Y 349.549,Z 366.564,A -85,B 0,C 180,E1 -13784.556,E2 -13784.556} C_VEL
LIN {X 0,Y 350.822,Z 358.726,A -85,B 0,C 180,E1 -13786.023,E2 -13786.023} C_VEL
LIN {X 0,Y 352.587,Z 348.866,A -85,B 0,C 180,E1 -13787.547,E2 -13787.547} C_VEL
LIN {X 0,Y 354.502,Z 337.834,A -85,B 0,C 180,E1 -13788.944,E2 -13788.944} C_VEL
LIN {X 0,Y 355.37,Z 330.344,A -85,B 0,C 180,E1 -13789.781,E2 -13789.781} C_VEL
LIN {X 0,Y 355.486,Z 321.503,A -85,B 0,C 180,E1 -13790.72,E2 -13790.72} C_VEL
LIN {X 0,Y 354.146,Z 308.989,A -85,B 0,C 180,E1 -13792.002,E2 -13792.002} C_VEL
LIN {X 0,Y 351.664,Z 297.414,A -85,B 0,C 180,E1 -13793.174,E2 -13793.174} C_VEL
LIN {X 0,Y 348.841,Z 288.176,A -85,B 0,C 180,E1 -13794.137,E2 -13794.137} C_VEL
LIN {X 0,Y 347.842,Z 284.47,A -85,B 0,C 180,E1 -13794.514,E2 -13794.514} C_VEL
LIN {X 0,Y 348.538,Z 279.138,A -85,B 0,C 180,E1 -13797.632,E2 -13797.632} C_VEL
LIN {X 0,Y 349.583,Z 273.076,A -85,B 0,C 180,E1 -13801.514,E2 -13801.514} C_VEL
LIN {X 0,Y 350.538,Z 268.646,A -85,B 0,C 180,E1 -13804.713,E2 -13804.713} C_VEL
LIN {X 0,Y 350.926,Z 265.992,A -85,B 0,C 180,E1 -13806.928,E2 -13806.928} C_VEL
LIN {X 0,Y 350.952,Z 264.201,A -85,B 0,C 180,E1 -13808.648,E2 -13808.648} C_VEL
LIN {X 0,Y 350.665,Z 261.802,A -85,B 0,C 180,E1 -13811.406,E2 -13811.406} C_VEL
LIN {X 0,Y 350.32,Z 259.674,A -85,B 0,C 180,E1 -13814.601,E2 -13814.601} C_VEL
LIN {X 0,Y 350.134,Z 258.524,A -85,B 0,C 180,E1 -13816.964,E2 -13816.964} C_VEL
LIN {X 0,Y 349.894,Z 257.555,A -85,B 0,C 180,E1 -13820.002,E2 -13820.002} C_VEL
LIN {X 0,Y 349.686,Z 257.094,A -85,B 0,C 180,E1 -13823.507,E2 -13823.507} C_VEL
LIN {X 0,Y 349.469,Z 257.152,A -85,B 0,C 180,E1 -13825.73,E2 -13825.73} C_VEL
LIN {X 0,Y 349.039,Z 257.581,A -85,B 0,C 180,E1 -13828.432,E2 -13828.432} C_VEL
LIN {X 0,Y 348.701,Z 258.271,A -85,B 0,C 180,E1 -13831.072,E2 -13831.072} C_VEL
LIN {X 0,Y 348.219,Z 259.726,A -85,B 0,C 180,E1 -13834.923,E2 -13834.923} C_VEL
LIN {X 0,Y 348.081,Z 260.712,A -85,B 0,C 180,E1 -13836.716,E2 -13836.716} C_VEL
LIN {X 0,Y 349.076,Z 263.36,A -85,B 0,C 180,E1 -13837.037,E2 -13837.037} C_VEL
LIN {X 0,Y 353.51,Z 272.401,A -85,B 0,C 180,E1 -13838.309,E2 -13838.309} C_VEL
LIN {X 0,Y 357.2,Z 282.642,A -85,B 0,C 180,E1 -13839.655,E2 -13839.655} C_VEL
LIN {X 0,Y 358.992,Z 289.703,A -85,B 0,C 180,E1 -13840.561,E2 -13840.561} C_VEL
LIN {X 0,Y 358.881,Z 292.325,A -85,B 0,C 180,E1 -13840.83,E2 -13840.83} C_VEL
LIN {X 0,Y 357.108,Z 304.306,A -85,B 0,C 180,E1 -13842.091,E2 -13842.091} C_VEL
LIN {X 0,Y 355.402,Z 313.986,A -85,B 0,C 180,E1 -13843.337,E2 -13843.337} C_VEL
LIN {X 0,Y 353.464,Z 324.546,A -85,B 0,C 180,E1 -13845.02,E2 -13845.02} C_VEL
LIN {X 0,Y 351.798,Z 333.117,A -85,B 0,C 180,E1 -13846.718,E2 -13846.718} C_VEL
LIN {X 0,Y 350.161,Z 341.135,A -85,B 0,C 180,E1 -13848.715,E2 -13848.715} C_VEL
LIN {X 0,Y 348.935,Z 347.375,A -85,B 0,C 180,E1 -13850.728,E2 -13850.728} C_VEL
LIN {X 0,Y 348.028,Z 351.511,A -85,B 0,C 180,E1 -13852.458,E2 -13852.458} C_VEL
LIN {X 0,Y 347.578,Z 354.6,A -85,B 0,C 180,E1 -13854.198,E2 -13854.198} C_VEL
LIN {X 0,Y 347.257,Z 356.119,A -85,B 0,C 180,E1 -13855.357,E2 -13855.357} C_VEL
LIN {X 0,Y 347.114,Z 357.23,A -85,B 0,C 180,E1 -13856.518,E2 -13856.518} C_VEL
LIN {X 0,Y 346.703,Z 357.979,A -85,B 0,C 180,E1 -13857.677,E2 -13857.677} C_VEL
LIN {X 0,Y 346.514,Z 358.269,A -85,B 0,C 180,E1 -13858.838,E2 -13858.838} C_VEL
LIN {X 0,Y 346.415,Z 357.652,A -85,B 0,C 180,E1 -13861.163,E2 -13861.163} C_VEL
LIN {X 0,Y 346.41,Z 356.739,A -85,B 0,C 180,E1 -13862.326,E2 -13862.326} C_VEL
LIN {X 0,Y 346.391,Z 355.374,A -85,B 0,C 180,E1 -13863.49,E2 -13863.49} C_VEL
LIN {X 0,Y 346.533,Z 352.539,A -85,B 0,C 180,E1 -13865.236,E2 -13865.236} C_VEL
LIN {X 0,Y 346.706,Z 348.533,A -85,B 0,C 180,E1 -13867.035,E2 -13867.035} C_VEL
LIN {X 0,Y 346.979,Z 343.634,A -85,B 0,C 180,E1 -13868.738,E2 -13868.738} C_VEL
LIN {X 0,Y 347.42,Z 337.323,A -85,B 0,C 180,E1 -13870.49,E2 -13870.49} C_VEL
LIN {X 0,Y 348.025,Z 329.516,A -85,B 0,C 180,E1 -13872.242,E2 -13872.242} C_VEL
LIN {X 0,Y 348.687,Z 321.576,A -85,B 0,C 180,E1 -13873.7,E2 -13873.7} C_VEL
LIN {X 0,Y 349.483,Z 310.91,A -85,B 0,C 180,E1 -13875.304,E2 -13875.304} C_VEL
LIN {X 0,Y 350.36,Z 300.238,A -85,B 0,C 180,E1 -13876.61,E2 -13876.61} C_VEL
LIN {X 0,Y 351.269,Z 288.44,A -85,B 0,C 180,E1 -13877.765,E2 -13877.765} C_VEL
LIN {X 0,Y 351.769,Z 280.462,A -85,B 0,C 180,E1 -13878.416,E2 -13878.416} C_VEL
LIN {X 0,Y 349.176,Z 266.734,A -85,B 0,C 180,E1 -13879.409,E2 -13879.409} C_VEL
LIN {X 0,Y 346.605,Z 253.295,A -85,B 0,C 180,E1 -13880.164,E2 -13880.164} C_VEL
LIN {X 0,Y 346.599,Z 249.354,A -85,B 0,C 180,E1 -13884.15,E2 -13884.15} C_VEL
LIN {X 0,Y 346.744,Z 246.692,A -85,B 0,C 180,E1 -13886.897,E2 -13886.897} C_VEL
LIN {X 0,Y 346.735,Z 245.846,A -85,B 0,C 180,E1 -13887.787,E2 -13887.787} C_VEL
LIN {X 0,Y 346.895,Z 245.277,A -85,B 0,C 180,E1 -13889.404,E2 -13889.404} C_VEL
LIN {X 0,Y 347.322,Z 245.222,A -85,B 0,C 180,E1 -13893.117,E2 -13893.117} C_VEL
LIN {X 0,Y 347.666,Z 245.176,A -85,B 0,C 180,E1 -13896.041,E2 -13896.041} C_VEL
LIN {X 0,Y 347.75,Z 245.167,A -85,B 0,C 180,E1 -13898.793,E2 -13898.793} C_VEL
LIN {X 0,Y 347.754,Z 245.165,A -85,B 0,C 180,E1 -13901.83,E2 -13901.83} C_VEL
LIN {X 0,Y 347.709,Z 245.175,A -85,B 0,C 180,E1 -13905.027,E2 -13905.027} C_VEL
LIN {X 0,Y 347.744,Z 245.167,A -85,B 0,C 180,E1 -13908.399,E2 -13908.399} C_VEL
LIN {X 0,Y 347.757,Z 245.168,A -85,B 0,C 180,E1 -13912.678,E2 -13912.678} C_VEL
LIN {X 0,Y 347.751,Z 245.165,A -85,B 0,C 180,E1 -13915.956,E2 -13915.956} C_VEL
LIN {X 0,Y 347.748,Z 245.165,A -85,B 0,C 180,E1 -13919.652,E2 -13919.652} C_VEL
LIN {X 0,Y 347.787,Z 245.16,A -85,B 0,C 180,E1 -13923.604,E2 -13923.604} C_VEL
LIN {X 0,Y 347.787,Z 245.164,A -85,B 0,C 180,E1 -13926.161,E2 -13926.161} C_VEL
LIN {X 0,Y 347.81,Z 245.16,A -85,B 0,C 180,E1 -13929.909,E2 -13929.909} C_VEL
LIN {X 0,Y 347.87,Z 245.155,A -85,B 0,C 180,E1 -13932.359,E2 -13932.359} C_VEL
LIN {X 0,Y 347.901,Z 245.151,A -85,B 0,C 180,E1 -13935.971,E2 -13935.971} C_VEL
LIN {X 0,Y 347.899,Z 245.148,A -85,B 0,C 180,E1 -13939.524,E2 -13939.524} C_VEL
LIN {X 0,Y 348.054,Z 245.127,A -85,B 0,C 180,E1 -13943.041,E2 -13943.041} C_VEL
LIN {X 0,Y 348.183,Z 245.116,A -85,B 0,C 180,E1 -13947.686,E2 -13947.686} C_VEL
LIN {X 0,Y 348.121,Z 245.12,A -85,B 0,C 180,E1 -13951.157,E2 -13951.157} C_VEL
LIN {X 0,Y 348.19,Z 245.111,A -85,B 0,C 180,E1 -13952.313,E2 -13952.313} C_VEL
LIN {X 0,Y 347.806,Z 245.289,A -85,B 0,C 180,E1 -13954.781,E2 -13954.781} C_VEL
LIN {X 0,Y 347.824,Z 249.424,A -85,B 0,C 180,E1 -13956.963,E2 -13956.963} C_VEL
LIN {X 0,Y 347.584,Z 256.186,A -85,B 0,C 180,E1 -13960.485,E2 -13960.485} C_VEL
LIN {X 0,Y 347.503,Z 260.72,A -85,B 0,C 180,E1 -13962.854,E2 -13962.854} C_VEL
LIN {X 0,Y 347.266,Z 267.586,A -85,B 0,C 180,E1 -13966.459,E2 -13966.459} C_VEL
LIN {X 0,Y 347.133,Z 273.424,A -85,B 0,C 180,E1 -13969.515,E2 -13969.515} C_VEL
LIN {X 0,Y 347.032,Z 276.608,A -85,B 0,C 180,E1 -13971.184,E2 -13971.184} C_VEL
LIN {X 0,Y 348.908,Z 286.426,A -85,B 0,C 180,E1 -13971.684,E2 -13971.684} C_VEL
LIN {X 0,Y 350.596,Z 296.83,A -85,B 0,C 180,E1 -13972.388,E2 -13972.388} C_VEL
LIN {X 0,Y 350.342,Z 306.09,A -85,B 0,C 180,E1 -13973.137,E2 -13973.137} C_VEL
LIN {X 0,Y 349.696,Z 315.918,A -85,B 0,C 180,E1 -13974.173,E2 -13974.173} C_VEL
LIN {X 0,Y 349.138,Z 322.817,A -85,B 0,C 180,E1 -13975.064,E2 -13975.064} C_VEL
LIN {X 0,Y 348.659,Z 328.928,A -85,B 0,C 180,E1 -13976.003,E2 -13976.003} C_VEL
LIN {X 0,Y 348.057,Z 335.973,A -85,B 0,C 180,E1 -13977.32,E2 -13977.32} C_VEL
LIN {X 0,Y 347.523,Z 341.966,A -85,B 0,C 180,E1 -13978.705,E2 -13978.705} C_VEL
LIN {X 0,Y 347.031,Z 347.8,A -85,B 0,C 180,E1 -13980.417,E2 -13980.417} C_VEL
LIN {X 0,Y 346.719,Z 351.365,A -85,B 0,C 180,E1 -13981.804,E2 -13981.804} C_VEL
LIN {X 0,Y 346.378,Z 354.797,A -85,B 0,C 180,E1 -13983.706,E2 -13983.706} C_VEL
LIN {X 0,Y 346.277,Z 356.035,A -85,B 0,C 180,E1 -13984.631,E2 -13984.631} C_VEL
LIN {X 0,Y 346.175,Z 357.207,A -85,B 0,C 180,E1 -13986.069,E2 -13986.069} C_VEL
LIN {X 0,Y 346.193,Z 357.582,A -85,B 0,C 180,E1 -13987.652,E2 -13987.652} C_VEL
LIN {X 0,Y 346.296,Z 356.796,A -85,B 0,C 180,E1 -13989.538,E2 -13989.538} C_VEL
LIN {X 0,Y 346.488,Z 355.637,A -85,B 0,C 180,E1 -13990.745,E2 -13990.745} C_VEL
LIN {X 0,Y 346.919,Z 352.725,A -85,B 0,C 180,E1 -13992.585,E2 -13992.585} C_VEL
LIN {X 0,Y 347.358,Z 348.963,A -85,B 0,C 180,E1 -13994.223,E2 -13994.223} C_VEL
LIN {X 0,Y 347.807,Z 345.159,A -85,B 0,C 180,E1 -13995.479,E2 -13995.479} C_VEL
LIN {X 0,Y 347.513,Z 342.299,A -85,B 0,C 180,E1 -13996.332,E2 -13996.332} C_VEL
LIN {X 0,Y 345.336,Z 337.232,A -85,B 0,C 180,E1 -13997.699,E2 -13997.699} C_VEL
LIN {X 0,Y 343.234,Z 331.363,A -85,B 0,C 180,E1 -13998.982,E2 -13998.982} C_VEL
LIN {X 0,Y 343.046,Z 327.251,A -85,B 0,C 180,E1 -13999.688,E2 -13999.688} C_VEL
LIN {X 0,Y 343.841,Z 319.442,A -85,B 0,C 180,E1 -14000.806,E2 -14000.806} C_VEL
LIN {X 0,Y 344.576,Z 311.381,A -85,B 0,C 180,E1 -14001.744,E2 -14001.744} C_VEL
LIN {X 0,Y 345.276,Z 302.783,A -85,B 0,C 180,E1 -14002.546,E2 -14002.546} C_VEL
LIN {X 0,Y 344.534,Z 295.933,A -85,B 0,C 180,E1 -14003.132,E2 -14003.132} C_VEL
LIN {X 0,Y 342.575,Z 286.323,A -85,B 0,C 180,E1 -14003.845,E2 -14003.845} C_VEL
LIN {X 0,Y 340.507,Z 277.955,A -85,B 0,C 180,E1 -14004.367,E2 -14004.367} C_VEL
LIN {X 0,Y 340.76,Z 270.411,A -85,B 0,C 180,E1 -14008.362,E2 -14008.362} C_VEL
LIN {X 0,Y 340.948,Z 264.095,A -85,B 0,C 180,E1 -14011.699,E2 -14011.699} C_VEL
LIN {X 0,Y 341.239,Z 256.579,A -85,B 0,C 180,E1 -14015.675,E2 -14015.675} C_VEL
LIN {X 0,Y 341.397,Z 251.551,A -85,B 0,C 180,E1 -14018.25,E2 -14018.25} C_VEL
LIN {X 0,Y 341.121,Z 248.026,A -85,B 0,C 180,E1 -14020.126,E2 -14020.126} C_VEL
LIN {X 0,Y 340.799,Z 246.036,A -85,B 0,C 180,E1 -14021.226,E2 -14021.226} C_VEL
LIN {X 0,Y 340.821,Z 246.032,A -85,B 0,C 180,E1 -14024.45,E2 -14024.45} C_VEL
LIN {X 0,Y 340.853,Z 246.032,A -85,B 0,C 180,E1 -14028.101,E2 -14028.101} C_VEL
LIN {X 0,Y 341.001,Z 246.011,A -85,B 0,C 180,E1 -14031.705,E2 -14031.705} C_VEL
LIN {X 0,Y 341.023,Z 246.007,A -85,B 0,C 180,E1 -14034.085,E2 -14034.085} C_VEL
LIN {X 0,Y 341.17,Z 245.988,A -85,B 0,C 180,E1 -14037.639,E2 -14037.639} C_VEL
LIN {X 0,Y 341.297,Z 245.972,A -85,B 0,C 180,E1 -14040,E2 -14040} C_VEL
LIN {X 0,Y 341.17,Z 245.989,A -85,B 0,C 180,E1 -14042.361,E2 -14042.361} C_VEL
LIN {X 0,Y 341.018,Z 246.008,A -85,B 0,C 180,E1 -14047.103,E2 -14047.103} C_VEL
LIN {X 0,Y 340.873,Z 246.024,A -85,B 0,C 180,E1 -14050.694,E2 -14050.694} C_VEL
LIN {X 0,Y 340.865,Z 246.026,A -85,B 0,C 180,E1 -14054.325,E2 -14054.325} C_VEL
LIN {X 0,Y 340.838,Z 246.027,A -85,B 0,C 180,E1 -14058.466,E2 -14058.466} C_VEL
LIN {X 0,Y 340.719,Z 246.043,A -85,B 0,C 180,E1 -14061.842,E2 -14061.842} C_VEL
LIN {X 0,Y 340.773,Z 246.038,A -85,B 0,C 180,E1 -14065.664,E2 -14065.664} C_VEL
LIN {X 0,Y 340.742,Z 246.042,A -85,B 0,C 180,E1 -14068.319,E2 -14068.319} C_VEL
LIN {X 0,Y 340.705,Z 246.046,A -85,B 0,C 180,E1 -14071.044,E2 -14071.044} C_VEL
LIN {X 0,Y 340.719,Z 246.042,A -85,B 0,C 180,E1 -14075.279,E2 -14075.279} C_VEL
LIN {X 0,Y 340.711,Z 246.046,A -85,B 0,C 180,E1 -14078.386,E2 -14078.386} C_VEL
LIN {X 0,Y 340.7,Z 246.044,A -85,B 0,C 180,E1 -14082.045,E2 -14082.045} C_VEL
LIN {X 0,Y 340.767,Z 246.167,A -85,B 0,C 180,E1 -14085.581,E2 -14085.581} C_VEL
LIN {X 0,Y 341.663,Z 251.285,A -85,B 0,C 180,E1 -14088.834,E2 -14088.834} C_VEL
LIN {X 0,Y 342.584,Z 256.49,A -85,B 0,C 180,E1 -14092.016,E2 -14092.016} C_VEL
LIN {X 0,Y 342.793,Z 260.327,A -85,B 0,C 180,E1 -14094.246,E2 -14094.246} C_VEL
LIN {X 0,Y 342.39,Z 264.067,A -85,B 0,C 180,E1 -14096.344,E2 -14096.344} C_VEL
LIN {X 0,Y 341.401,Z 271.496,A -85,B 0,C 180,E1 -14100.392,E2 -14100.392} C_VEL
LIN {X 0,Y 340.659,Z 278.852,A -85,B 0,C 180,E1 -14104.326,E2 -14104.326} C_VEL
LIN {X 0,Y 339.993,Z 286.72,A -85,B 0,C 180,E1 -14108.465,E2 -14108.465} C_VEL
LIN {X 0,Y 339.749,Z 290.577,A -85,B 0,C 180,E1 -14110.476,E2 -14110.476} C_VEL
LIN {X 0,Y 341.121,Z 304.022,A -85,B 0,C 180,E1 -14111.162,E2 -14111.162} C_VEL
LIN {X 0,Y 342.618,Z 317.493,A -85,B 0,C 180,E1 -14112.08,E2 -14112.08} C_VEL
LIN {X 0,Y 343.49,Z 327.148,A -85,B 0,C 180,E1 -14112.895,E2 -14112.895} C_VEL
LIN {X 0,Y 342.653,Z 338.963,A -85,B 0,C 180,E1 -14114.078,E2 -14114.078} C_VEL
LIN {X 0,Y 341.626,Z 349.55,A -85,B 0,C 180,E1 -14115.39,E2 -14115.39} C_VEL
LIN {X 0,Y 340.641,Z 363.245,A -85,B 0,C 180,E1 -14117.489,E2 -14117.489} C_VEL
LIN {X 0,Y 340.031,Z 371.491,A -85,B 0,C 180,E1 -14118.978,E2 -14118.978} C_VEL
LIN {X 0,Y 339.663,Z 377.991,A -85,B 0,C 180,E1 -14120.472,E2 -14120.472} C_VEL
LIN {X 0,Y 339.495,Z 382.257,A -85,B 0,C 180,E1 -14121.668,E2 -14121.668} C_VEL
LIN {X 0,Y 339.34,Z 385.79,A -85,B 0,C 180,E1 -14122.862,E2 -14122.862} C_VEL
LIN {X 0,Y 339.243,Z 389.862,A -85,B 0,C 180,E1 -14124.651,E2 -14124.651} C_VEL
LIN {X 0,Y 339.204,Z 392.666,A -85,B 0,C 180,E1 -14126.437,E2 -14126.437} C_VEL
LIN {X 0,Y 339.357,Z 394.738,A -85,B 0,C 180,E1 -14128.814,E2 -14128.814} C_VEL
LIN {X 0,Y 339.332,Z 395.438,A -85,B 0,C 180,E1 -14130,E2 -14130} C_VEL
LIN {X 0,Y 339.325,Z 395.696,A -85,B 0,C 180,E1 -14131.187,E2 -14131.187} C_VEL
LIN {X 0,Y 339.119,Z 394.975,A -85,B 0,C 180,E1 -14133.565,E2 -14133.565} C_VEL
LIN {X 0,Y 339.107,Z 393.977,A -85,B 0,C 180,E1 -14134.756,E2 -14134.756} C_VEL
LIN {X 0,Y 339.13,Z 392.55,A -85,B 0,C 180,E1 -14135.948,E2 -14135.948} C_VEL
LIN {X 0,Y 339.369,Z 389.633,A -85,B 0,C 180,E1 -14137.736,E2 -14137.736} C_VEL
LIN {X 0,Y 339.743,Z 385.716,A -85,B 0,C 180,E1 -14139.526,E2 -14139.526} C_VEL
LIN {X 0,Y 340.393,Z 380.722,A -85,B 0,C 180,E1 -14141.312,E2 -14141.312} C_VEL
LIN {X 0,Y 341.714,Z 373.407,A -85,B 0,C 180,E1 -14143.378,E2 -14143.378} C_VEL
LIN {X 0,Y 342.926,Z 365.695,A -85,B 0,C 180,E1 -14145.148,E2 -14145.148} C_VEL
LIN {X 0,Y 344.634,Z 356.292,A -85,B 0,C 180,E1 -14146.894,E2 -14146.894} C_VEL
LIN {X 0,Y 346.709,Z 345.904,A -85,B 0,C 180,E1 -14148.465,E2 -14148.465} C_VEL
LIN {X 0,Y 348.736,Z 334.467,A -85,B 0,C 180,E1 -14149.882,E2 -14149.882} C_VEL
LIN {X 0,Y 349.194,Z 323.935,A -85,B 0,C 180,E1 -14151.081,E2 -14151.081} C_VEL
LIN {X 0,Y 348.175,Z 311.851,A -85,B 0,C 180,E1 -14152.41,E2 -14152.41} C_VEL
LIN {X 0,Y 346.129,Z 301.265,A -85,B 0,C 180,E1 -14153.567,E2 -14153.567} C_VEL
LIN {X 0,Y 342.283,Z 288.007,A -85,B 0,C 180,E1 -14155.058,E2 -14155.058} C_VEL
LIN {X 0,Y 341.112,Z 284.518,A -85,B 0,C 180,E1 -14155.451,E2 -14155.451} C_VEL
LIN {X 0,Y 341.034,Z 283.773,A -85,B 0,C 180,E1 -14155.519,E2 -14155.519} C_VEL
LIN {X 0,Y 342.008,Z 277.295,A -85,B 0,C 180,E1 -14159.55,E2 -14159.55} C_VEL
LIN {X 0,Y 343.228,Z 271.55,A -85,B 0,C 180,E1 -14163.564,E2 -14163.564} C_VEL
LIN {X 0,Y 343.876,Z 268.109,A -85,B 0,C 180,E1 -14166.349,E2 -14166.349} C_VEL
LIN {X 0,Y 343.973,Z 265.321,A -85,B 0,C 180,E1 -14169.067,E2 -14169.067} C_VEL
LIN {X 0,Y 343.826,Z 263.774,A -85,B 0,C 180,E1 -14170.861,E2 -14170.861} C_VEL
LIN {X 0,Y 343.424,Z 261.454,A -85,B 0,C 180,E1 -14174.253,E2 -14174.253} C_VEL
LIN {X 0,Y 343.157,Z 259.89,A -85,B 0,C 180,E1 -14177.502,E2 -14177.502} C_VEL
LIN {X 0,Y 342.897,Z 258.885,A -85,B 0,C 180,E1 -14181.156,E2 -14181.156} C_VEL
LIN {X 0,Y 342.754,Z 258.628,A -85,B 0,C 180,E1 -14183.514,E2 -14183.514} C_VEL
LIN {X 0,Y 342.393,Z 258.72,A -85,B 0,C 180,E1 -14186.344,E2 -14186.344} C_VEL
LIN {X 0,Y 341.957,Z 259.294,A -85,B 0,C 180,E1 -14189.678,E2 -14189.678} C_VEL
LIN {X 0,Y 341.484,Z 260.331,A -85,B 0,C 180,E1 -14193.078,E2 -14193.078} C_VEL
LIN {X 0,Y 341.192,Z 261.368,A -85,B 0,C 180,E1 -14195.672,E2 -14195.672} C_VEL
LIN {X 0,Y 341.747,Z 263.219,A -85,B 0,C 180,E1 -14195.891,E2 -14195.891} C_VEL
LIN {X 0,Y 346.437,Z 272.398,A -85,B 0,C 180,E1 -14197.329,E2 -14197.329} C_VEL
LIN {X 0,Y 350.144,Z 281.774,A -85,B 0,C 180,E1 -14198.683,E2 -14198.683} C_VEL
LIN {X 0,Y 352.825,Z 291.798,A -85,B 0,C 180,E1 -14200.063,E2 -14200.063} C_VEL
LIN {X 0,Y 352.934,Z 292.977,A -85,B 0,C 180,E1 -14200.213,E2 -14200.213} C_VEL
LIN {X 0,Y 350.846,Z 305.835,A -85,B 0,C 180,E1 -14201.609,E2 -14201.609} C_VEL
LIN {X 0,Y 348.846,Z 316.205,A -85,B 0,C 180,E1 -14203.015,E2 -14203.015} C_VEL
LIN {X 0,Y 346.842,Z 326.409,A -85,B 0,C 180,E1 -14204.727,E2 -14204.727} C_VEL
LIN {X 0,Y 345.069,Z 334.671,A -85,B 0,C 180,E1 -14206.454,E2 -14206.454} C_VEL
LIN {X 0,Y 343.548,Z 341.441,A -85,B 0,C 180,E1 -14208.196,E2 -14208.196} C_VEL
LIN {X 0,Y 342.376,Z 347.073,A -85,B 0,C 180,E1 -14210.011,E2 -14210.011} C_VEL
LIN {X 0,Y 341.218,Z 351.266,A -85,B 0,C 180,E1 -14211.71,E2 -14211.71} C_VEL
LIN {X 0,Y 340.932,Z 353.547,A -85,B 0,C 180,E1 -14212.895,E2 -14212.895} C_VEL
LIN {X 0,Y 340.57,Z 355.391,A -85,B 0,C 180,E1 -14214.078,E2 -14214.078} C_VEL
LIN {X 0,Y 340.054,Z 357.884,A -85,B 0,C 180,E1 -14216.445,E2 -14216.445} C_VEL
LIN {X 0,Y 339.646,Z 358.518,A -85,B 0,C 180,E1 -14217.628,E2 -14217.628} C_VEL
LIN {X 0,Y 339.364,Z 358.561,A -85,B 0,C 180,E1 -14220,E2 -14220} C_VEL
LIN {X 0,Y 339.336,Z 357.986,A -85,B 0,C 180,E1 -14221.187,E2 -14221.187} C_VEL
LIN {X 0,Y 339.313,Z 356.964,A -85,B 0,C 180,E1 -14222.374,E2 -14222.374} C_VEL
LIN {X 0,Y 339.31,Z 355.534,A -85,B 0,C 180,E1 -14223.563,E2 -14223.563} C_VEL
LIN {X 0,Y 339.457,Z 352.577,A -85,B 0,C 180,E1 -14225.346,E2 -14225.346} C_VEL
LIN {X 0,Y 339.64,Z 348.571,A -85,B 0,C 180,E1 -14227.132,E2 -14227.132} C_VEL
LIN {X 0,Y 340.021,Z 342.444,A -85,B 0,C 180,E1 -14229.218,E2 -14229.218} C_VEL
LIN {X 0,Y 340.507,Z 335.706,A -85,B 0,C 180,E1 -14231.007,E2 -14231.007} C_VEL
LIN {X 0,Y 341.177,Z 327.391,A -85,B 0,C 180,E1 -14232.794,E2 -14232.794} C_VEL
LIN {X 0,Y 342.015,Z 317.679,A -85,B 0,C 180,E1 -14234.487,E2 -14234.487} C_VEL
LIN {X 0,Y 342.797,Z 306.438,A -85,B 0,C 180,E1 -14236.068,E2 -14236.068} C_VEL
LIN {X 0,Y 343.66,Z 296.095,A -85,B 0,C 180,E1 -14237.25,E2 -14237.25} C_VEL
LIN {X 0,Y 344.545,Z 284.957,A -85,B 0,C 180,E1 -14238.278,E2 -14238.278} C_VEL
LIN {X 0,Y 344.621,Z 280.247,A -85,B 0,C 180,E1 -14238.658,E2 -14238.658} C_VEL
LIN {X 0,Y 341.933,Z 266.228,A -85,B 0,C 180,E1 -14239.686,E2 -14239.686} C_VEL
LIN {X 0,Y 339.513,Z 253.652,A -85,B 0,C 180,E1 -14240.406,E2 -14240.406} C_VEL
LIN {X 0,Y 339.527,Z 249.69,A -85,B 0,C 180,E1 -14244.456,E2 -14244.456} C_VEL
LIN {X 0,Y 339.68,Z 247.095,A -85,B 0,C 180,E1 -14247.167,E2 -14247.167} C_VEL
LIN {X 0,Y 339.72,Z 246.171,A -85,B 0,C 180,E1 -14248.413,E2 -14248.413} C_VEL
LIN {X 0,Y 340.177,Z 246.108,A -85,B 0,C 180,E1 -14252.491,E2 -14252.491} C_VEL
LIN {X 0,Y 340.519,Z 246.071,A -85,B 0,C 180,E1 -14255.303,E2 -14255.303} C_VEL
LIN {X 0,Y 340.702,Z 246.043,A -85,B 0,C 180,E1 -14258.384,E2 -14258.384} C_VEL
LIN {X 0,Y 340.702,Z 246.043,A -85,B 0,C 180,E1 -14262.045,E2 -14262.045} C_VEL
LIN {X 0,Y 340.655,Z 246.049,A -85,B 0,C 180,E1 -14266.227,E2 -14266.227} C_VEL
LIN {X 0,Y 340.674,Z 246.05,A -85,B 0,C 180,E1 -14268.688,E2 -14268.688} C_VEL
LIN {X 0,Y 340.721,Z 246.04,A -85,B 0,C 180,E1 -14271.771,E2 -14271.771} C_VEL
LIN {X 0,Y 340.725,Z 246.04,A -85,B 0,C 180,E1 -14275.596,E2 -14275.596} C_VEL
LIN {X 0,Y 340.699,Z 246.046,A -85,B 0,C 180,E1 -14278.955,E2 -14278.955} C_VEL
LIN {X 0,Y 340.714,Z 246.047,A -85,B 0,C 180,E1 -14282.496,E2 -14282.496} C_VEL
LIN {X 0,Y 340.755,Z 246.036,A -85,B 0,C 180,E1 -14285.638,E2 -14285.638} C_VEL
LIN {X 0,Y 340.737,Z 246.039,A -85,B 0,C 180,E1 -14289.473,E2 -14289.473} C_VEL
LIN {X 0,Y 340.861,Z 246.026,A -85,B 0,C 180,E1 -14291.984,E2 -14291.984} C_VEL
LIN {X 0,Y 340.873,Z 246.023,A -85,B 0,C 180,E1 -14295.705,E2 -14295.705} C_VEL
LIN {X 0,Y 340.851,Z 246.025,A -85,B 0,C 180,E1 -14299.305,E2 -14299.305} C_VEL
LIN {X 0,Y 341.001,Z 246.005,A -85,B 0,C 180,E1 -14302.896,E2 -14302.896} C_VEL
LIN {X 0,Y 340.808,Z 246.03,A -85,B 0,C 180,E1 -14305.268,E2 -14305.268} C_VEL
LIN {X 0,Y 341.12,Z 245.995,A -85,B 0,C 180,E1 -14307.638,E2 -14307.638} C_VEL
LIN {X 0,Y 341.092,Z 245.995,A -85,B 0,C 180,E1 -14311.18,E2 -14311.18} C_VEL
LIN {X 0,Y 341.125,Z 245.99,A -85,B 0,C 180,E1 -14312.361,E2 -14312.361} C_VEL
LIN {X 0,Y 340.743,Z 246.066,A -85,B 0,C 180,E1 -14314.584,E2 -14314.584} C_VEL
LIN {X 0,Y 340.858,Z 249.662,A -85,B 0,C 180,E1 -14316.511,E2 -14316.511} C_VEL
LIN {X 0,Y 340.55,Z 257.616,A -85,B 0,C 180,E1 -14320.704,E2 -14320.704} C_VEL
LIN {X 0,Y 340.361,Z 264.521,A -85,B 0,C 180,E1 -14324.346,E2 -14324.346} C_VEL
LIN {X 0,Y 340.204,Z 271.704,A -85,B 0,C 180,E1 -14328.143,E2 -14328.143} C_VEL
LIN {X 0,Y 339.997,Z 276.957,A -85,B 0,C 180,E1 -14330.907,E2 -14330.907} C_VEL
LIN {X 0,Y 341.854,Z 286.557,A -85,B 0,C 180,E1 -14331.404,E2 -14331.404} C_VEL
LIN {X 0,Y 343.424,Z 296.277,A -85,B 0,C 180,E1 -14332.068,E2 -14332.068} C_VEL
LIN {X 0,Y 343.764,Z 300.012,A -85,B 0,C 180,E1 -14332.362,E2 -14332.362} C_VEL
LIN {X 0,Y 343.195,Z 309.519,A -85,B 0,C 180,E1 -14333.216,E2 -14333.216} C_VEL
LIN {X 0,Y 342.665,Z 317.049,A -85,B 0,C 180,E1 -14334.056,E2 -14334.056} C_VEL
LIN {X 0,Y 342.074,Z 324.519,A -85,B 0,C 180,E1 -14335.07,E2 -14335.07} C_VEL
LIN {X 0,Y 341.457,Z 331.758,A -85,B 0,C 180,E1 -14336.265,E2 -14336.265} C_VEL
LIN {X 0,Y 340.718,Z 339.652,A -85,B 0,C 180,E1 -14337.895,E2 -14337.895} C_VEL
LIN {X 0,Y 340.213,Z 345.182,A -85,B 0,C 180,E1 -14339.381,E2 -14339.381} C_VEL
LIN {X 0,Y 339.94,Z 348.45,A -85,B 0,C 180,E1 -14340.432,E2 -14340.432} C_VEL
LIN {X 0,Y 339.591,Z 352.146,A -85,B 0,C 180,E1 -14341.949,E2 -14341.949} C_VEL
LIN {X 0,Y 339.368,Z 354.625,A -85,B 0,C 180,E1 -14343.284,E2 -14343.284} C_VEL
LIN {X 0,Y 339.113,Z 357.124,A -85,B 0,C 180,E1 -14345.471,E2 -14345.471} C_VEL
LIN {X 0,Y 339.104,Z 357.853,A -85,B 0,C 180,E1 -14346.944,E2 -14346.944} C_VEL
LIN {X 0,Y 339.128,Z 357.806,A -85,B 0,C 180,E1 -14348.441,E2 -14348.441} C_VEL
LIN {X 0,Y 339.269,Z 356.943,A -85,B 0,C 180,E1 -14349.963,E2 -14349.963} C_VEL
LIN {X 0,Y 339.688,Z 354.737,A -85,B 0,C 180,E1 -14351.855,E2 -14351.855} C_VEL
LIN {X 0,Y 340.17,Z 351.156,A -85,B 0,C 180,E1 -14353.688,E2 -14353.688} C_VEL
LIN {X 0,Y 340.567,Z 347.666,A -85,B 0,C 180,E1 -14355.024,E2 -14355.024} C_VEL
LIN {X 0,Y 341.277,Z 341.971,A -85,B 0,C 180,E1 -14356.7,E2 -14356.7} C_VEL
LIN {X 0,Y 342.021,Z 335.734,A -85,B 0,C 180,E1 -14358.149,E2 -14358.149} C_VEL
LIN {X 0,Y 343.046,Z 327.251,A -85,B 0,C 180,E1 -14359.688,E2 -14359.688} C_VEL
LIN {X 0,Y 342.916,Z 323.071,A -85,B 0,C 180,E1 -14360.355,E2 -14360.355} C_VEL
LIN {X 0,Y 341.07,Z 315.894,A -85,B 0,C 180,E1 -14361.437,E2 -14361.437} C_VEL
LIN {X 0,Y 339.061,Z 308.084,A -85,B 0,C 180,E1 -14362.438,E2 -14362.438} C_VEL
LIN {X 0,Y 338.539,Z 302.937,A -85,B 0,C 180,E1 -14362.945,E2 -14362.945} C_VEL
LIN {X 0,Y 337.156,Z 293.661,A -85,B 0,C 180,E1 -14363.758,E2 -14363.758} C_VEL
LIN {X 0,Y 334.479,Z 282.075,A -85,B 0,C 180,E1 -14364.573,E2 -14364.573} C_VEL
LIN {X 0,Y 333.52,Z 278.337,A -85,B 0,C 180,E1 -14364.797,E2 -14364.797} C_VEL
LIN {X 0,Y 333.778,Z 270.615,A -85,B 0,C 180,E1 -14368.944,E2 -14368.944} C_VEL
LIN {X 0,Y 334.019,Z 264.07,A -85,B 0,C 180,E1 -14372.426,E2 -14372.426} C_VEL
LIN {X 0,Y 334.339,Z 256.532,A -85,B 0,C 180,E1 -14376.46,E2 -14376.46} C_VEL
LIN {X 0,Y 334.422,Z 251.66,A -85,B 0,C 180,E1 -14379.068,E2 -14379.068} C_VEL
LIN {X 0,Y 333.76,Z 246.913,A -85,B 0,C 180,E1 -14381.667,E2 -14381.667} C_VEL
LIN {X 0,Y 333.81,Z 246.906,A -85,B 0,C 180,E1 -14385.576,E2 -14385.576} C_VEL
LIN {X 0,Y 333.836,Z 246.905,A -85,B 0,C 180,E1 -14389.078,E2 -14389.078} C_VEL
LIN {X 0,Y 333.973,Z 246.885,A -85,B 0,C 180,E1 -14392.746,E2 -14392.746} C_VEL
LIN {X 0,Y 333.804,Z 246.908,A -85,B 0,C 180,E1 -14395.169,E2 -14395.169} C_VEL
LIN {X 0,Y 334.107,Z 246.868,A -85,B 0,C 180,E1 -14397.589,E2 -14397.589} C_VEL
LIN {X 0,Y 334.248,Z 246.85,A -85,B 0,C 180,E1 -14400,E2 -14400} C_VEL
